// init traj filter
m_jnt3OTG.init(m_cmdJntPos[3], 0, m_retractVel, m_retractAcc, g_slaveArmCtrlCycleTime);

// set wait time before start retract
IF SlaveArmControl.m_slaveRobot.m_lastSlaveArmState[i_slaveArm.armIdx] = SlaveArmState_PanelReady THEN
	m_waitTime := 0;
ELSE
	m_waitTime :=1.0;
END_IF

// decide instrument joint zero position and init traj filter
FOR i:=1 TO 5 DO
	cycleNum := FLOOR(i_slaveArm.curJntPos[i+3]/g_2pi);
	m_instruJntTargetPos[i]:=cycleNum* g_2Pi;
	m_instruJntOTG[i].init(m_cmdJntPos[i+3], 0,m_instruJntVel, m_instruJntAcc, g_slaveArmCtrlCycleTime);
END_FOR

// update commands to arm
copyCmds(r_slaveArmCtrlCmd);
END_METHOD

END_FUNCTION_BLOCK

// ---- FBs_SlaveControllers/FB_SlaveCtrlInstruInvasion.TcPOU
// Brief: Slave Arm Invase instrument to record position
FUNCTION_BLOCK PUBLIC FB_SlaveCtrlInstruInvasion EXTENDS FB_SlaveArmCtrlBase
VAR_INPUT
END_VAR
VAR_OUTPUT
END_VAR
VAR
	// invasion buffer
	m_instruInvasionDepthSafetyBuffer :LREAL:= 0.01;
		
	// max damping when reaching invasion depth
	m_maxDamp :LREAL :=500;
	
	// current distance form target invasion depth 
	m_invasionDis :LREAL :=0;
	
	// distance threshold from target depth to start enable damp
	m_dampDisThres :LREAL :=0.03;
	
END_VAR

// override this function in each exact controller
METHOD PROTECTED calcCmdJntPos : BOOL
VAR_IN_OUT CONSTANT
	i_endoscopePose : ST_Frame;
	i_masterStatus :ST_MasterStatus;
	i_setupStatus: ST_SetupStatus;
	i_slaveArm :FB_SlaveArm;
END_VAR

VAR 
	curInstruDepth:LREAL;
END_VAR
m_cmdJntPos[3]:=i_slaveArm.curJntPos[3];
// compute current instrument depth
curInstruDepth := i_slaveArm.curJntPos[3]-i_slaveArm.instrument.instruTypeInfo.m_rodLength-i_slaveArm.instrument.instruTypeInfo.m_headLength
						- i_slaveArm.instrument.instruTypeInfo.m_fingerLength-m_instruInvasionDepthSafetyBuffer;

m_invasionDis:=curInstruDepth-i_slaveArm.m_instruInvasionDepth;
						
m_isFinished := curInstruDepth<= i_slaveArm.m_instruInvasionDepth;
END_METHOD

// override this function in each exact controller
METHOD PROTECTED calcCmdJntTrq : BOOL
VAR_IN_OUT CONSTANT
	i_endoscopePose : ST_Frame;
	i_masterStatus :ST_MasterStatus;
	i_setupStatus: ST_SetupStatus;
	i_slaveArm :FB_SlaveArm;
END_VAR
VAR
	dampScale :lreal ;
END_VAR
// set joint torque to zero in default
m_cmdJntTrq := g_zeroVec8d;

dampScale  :=LIMIT(0, 1-m_invasionDis/m_dampDisThres,1);
m_cmdJntTrq[3]:= -dampScale * m_maxDamp * i_slaveArm.curJntVel[3];
END_METHOD

METHOD PUBLIC init : BOOL
VAR_IN_OUT CONSTANT
	i_slaveArm	:FB_SlaveArm;
END_VAR
VAR_IN_OUT 
	r_slaveArmCtrlCmd :ST_SlaveArmCtrlCmds;
END_VAR
// check if to hold the command joint position unchanged
m_holdLastCmds := checkToHoldLastCmds(i_slaveArm);

//init
SUPER^.Init(i_slaveArm,r_slaveArmCtrlCmd);
m_invasionDis:=m_dampDisThres;

// only joint 3 is allowed to be pushed
m_jntOPMode := g_slaveAllPosMode;
m_jntOPMode[3]:=DriverOPMode_Trq;

// update commands to arm
copyCmds(r_slaveArmCtrlCmd);
END_METHOD

END_FUNCTION_BLOCK

// ---- FBs_SlaveControllers/FB_SlaveCtrlDisable.TcPOU
// Brief: Disable a Slave Arm 
FUNCTION_BLOCK PUBLIC FB_SlaveCtrlDisable EXTENDS FB_SlaveArmCtrlBase
VAR_INPUT
END_VAR
VAR_OUTPUT
END_VAR
VAR
END_VAR

// override this function in each exact controller
METHOD PROTECTED calcCmdJntPos : BOOL
VAR_IN_OUT CONSTANT
	// endoscope pose in cart coordinate
	i_endoscopePose : ST_Frame;
	
	// master arm data
	i_masterStatus :ST_MasterStatus;
	
	// setup arm data
	i_setupStatus: ST_SetupStatus;
	
	// slave arm data
	i_slaveArm :FB_SlaveArm;
END_VAR
m_cmdJntPos := i_slaveArm.curJntPos;
END_METHOD

// override this function in each exact controller
// NOTICE: set joint control mode here, and do some initialization if needed
METHOD PUBLIC init : BOOL
VAR_IN_OUT CONSTANT
	i_slaveArm	:FB_SlaveArm;
END_VAR
VAR_IN_OUT 
	r_slaveArmCtrlCmd :ST_SlaveArmCtrlCmds;
END_VAR


VAR
	i:INT;
END_VAR
SUPER^.Init(i_slaveArm,r_slaveArmCtrlCmd);

// disable all joints
 m_jntEnableFlag :=g_zeroVec8i;
 
 // update commands to arm
copyCmds(r_slaveArmCtrlCmd);
END_METHOD

END_FUNCTION_BLOCK

// ---- FBs_SlaveControllers/FB_SlaveCtrlInstruCali.TcPOU
// Brief: Calibrate the zero position of Instrument
FUNCTION_BLOCK PUBLIC FB_SlaveCtrlInstruCali EXTENDS FB_SlaveArmCtrlBase
VAR
	// mount motion planning
	m_jntOTG :ARRAY[1..8] OF FB_secOrdTrajFilter;
	m_instruMountVel :LREAL := 1*PI;
	m_instruMountAcc :LREAL := 2*PI;
	
	// 	cali status
	m_rollJntCaliStatus :INT := 0;
	m_pitchJntCaliStatus :INT := 0;
	m_yawJntCaliStatus :INT := 0;
	
	// flag if zero position is written to CoE
	m_zeroPosWritten :BOOL;
	
	// joint current threshold which indicate panel is buckled with instrument
	m_maxJntCurrent :LREAL := 100;
	
	// joint current threshold which indicate finger closed
	m_fingerCloseCurrent :LREAL := 50;
	
	// joint position at limits
	m_jntLimitPos1, m_jntLimitPos2, m_jntCaliPos :LREAL;
	m_jntLimitPos3, m_jntLimitPos4 :LREAL;

	// flag if joint is mounted
	m_jointMounted :ARRAY[1..8] OF BOOL := [5(FALSE)];
	
	// instrument mount motion range
	m_mountMotionAng :LREAL :=30*g_deg2Rad;
	
	// command mount motion
	m_targetMountPos :Vec8d;
	
	// instrument zero position
	m_instruZeroPosition :Vec5d;
	
	// angle to close finger
	m_baseCloseAngle :LREAL := 1*g_deg2Rad;
	m_bipolarCloseAngle :LREAL := 5*g_deg2Rad;
	m_proGraspCloseAngle:LREAL := 25*g_deg2Rad;
	
END_VAR

// override this function in each exact controller
METHOD PROTECTED calcCmdJntPos : BOOL
VAR_IN_OUT CONSTANT
	i_endoscopePose : ST_Frame;
	i_masterStatus :ST_MasterStatus;
	i_setupStatus: ST_SetupStatus;
	i_slaveArm :FB_SlaveArm;
END_VAR

VAR 
	i :INT;
END_VAR
// retur directly if instrument/endoscope is not readed
IF NOT i_slaveArm.instrument.onChipData.m_InstruReadSucceed THEN
	m_rollJntCaliStatus :=0;
	m_pitchJntCaliStatus :=0;
	m_yawJntCaliStatus :=0;
	m_zeroPosWritten :=FALSE;
	FOR i:=4 TO 8 DO
		m_jointMounted[i]:=FALSE;
	END_FOR
	return;
END_IF

// write zero position to CoE
IF m_yawJntCaliStatus = -1 THEN
	IF   NOT m_zeroPosWritten THEN
		m_zeroPosWritten := i_slaveArm.instrument.writeZeroPosToChip(m_instruZeroPosition[1],m_instruZeroPosition[2],m_instruZeroPosition[3]);
	END_IF
	RETURN;
END_IF;

// move joint to zero position
IF m_rollJntCaliStatus <> -1 THEN
	rollJntCali(i_slaveArm);
ELSIF m_pitchJntCaliStatus <> -1 THEN
	pitchJntCali(i_slaveArm);
ELSIF m_yawJntCaliStatus <> -1 THEN
	IF  i_slaveArm.instrument.InstruTypeInfo.m_isSingleFinger THEN
		yawJntCali_finger(i_slaveArm);
	ELSE
		yawJntCali_gripper(i_slaveArm);
	END_IF

END_IF

IF m_yawJntCaliStatus = -1 THEN
	FOR  i:=1 TO  5 DO
		m_instruZeroPosition[i]:=i_slaveArm.linkSingle[i+3];
	END_FOR
END_IF
END_METHOD

METHOD PUBLIC init : BOOL
VAR_IN_OUT CONSTANT
	i_slaveArm	:FB_SlaveArm;
END_VAR
VAR_IN_OUT 
	r_slaveArmCtrlCmd :ST_SlaveArmCtrlCmds;
END_VAR

VAR
	i : INT;
END_VAR
// check if to hold the command joint position unchanged
m_holdLastCmds := checkToHoldLastCmds(i_slaveArm);

SUPER^.Init(i_slaveArm,r_slaveArmCtrlCmd);
m_jntOPMode[4] := DriverOPMode_PosTrq;
m_jntOPMode[5] := DriverOPMode_PosTrq;
m_jntOPMode[6] := DriverOPMode_PosTrq;
m_jntOPMode[7] := DriverOPMode_PosTrq;
m_jntOPMode[8] := DriverOPMode_PosTrq;

FOR i:=4 TO 8 DO
	m_targetMountPos[i]:=m_cmdJntPos[i];
	m_jntOTG[i].init(m_targetMountPos[i], 0,m_instruMountVel, m_instruMountAcc, g_slaveArmCtrlCycleTime);
	m_jointMounted[i]:=FALSE;
END_FOR

m_rollJntCaliStatus :=0;
m_pitchJntCaliStatus :=0;
m_yawJntCaliStatus :=0;
m_zeroPosWritten := false;

// update commands to arm
copyCmds(r_slaveArmCtrlCmd);
END_METHOD

METHOD pitchJntCali : BOOL
VAR_IN_OUT CONSTANT
	i_slaveArm :FB_SlaveArm;
END_VAR

VAR 
	i :INT;
	curJntPos :Vec8d;
	jntIdx :INT;
END_VAR
jntIdx:=6;
curJntPos := i_slaveArm.curJntPos;

CASE m_pitchJntCaliStatus OF
	// rotate clockwise
	0:
		m_targetMountPos[jntIdx]:=curJntPos[jntIdx]+m_mountMotionAng;
	
		//buckle joint
		IF i_slaveArm.filtJntCurrent[jntIdx]> m_maxJntCurrent THEN 
			m_jntLimitPos1 := curJntPos[jntIdx];
			m_targetMountPos[jntIdx]:=curJntPos[jntIdx];
			m_jntOTG[jntIdx].init(m_targetMountPos[jntIdx], 0,m_instruMountVel, m_instruMountAcc, g_slaveArmCtrlCycleTime);
			m_pitchJntCaliStatus := 1;
		END_IF
		
	// rotate anticlockwise
	1:
		m_targetMountPos[jntIdx]:=curJntPos[jntIdx]-m_mountMotionAng;
	
		//buckle  joint
		IF i_slaveArm.filtJntCurrent[jntIdx]<- m_maxJntCurrent THEN 
			m_jntLimitPos2 := curJntPos[jntIdx];
			m_targetMountPos[jntIdx]:=curJntPos[jntIdx];
			m_jntOTG[jntIdx].init(m_targetMountPos[jntIdx], 0,m_instruMountVel, m_instruMountAcc, g_slaveArmCtrlCycleTime);
			m_pitchJntCaliStatus := 2;
		END_IF
	
	2:// calculate center/calibarted position
		m_targetMountPos[jntIdx] :=  (m_jntLimitPos1 + m_jntLimitPos2)/2+ i_slaveArm.instrument.instruTypeInfo.m_instruPitchBachlash/2.0;
		m_pitchJntCaliStatus := 3;

	3:
		IF ABS(m_targetMountPos[jntIdx]-curJntPos[jntIdx]) <GVL_SlaveControlParameters.g_jntCtrlAngTolHigh  THEN
			m_pitchJntCaliStatus := -1;
		END_IF
		
END_CASE

// traj plan
m_jntOTG[jntIdx].run(m_targetMountPos[jntIdx],0.0, o_cmdAcc=>m_cmdJntAcc[jntIdx],o_cmdVel=>m_cmdJntVel[jntIdx],o_cmdPos=>m_cmdJntPos[jntIdx]);
END_METHOD

METHOD rollJntCali : BOOL
VAR_IN_OUT CONSTANT
	i_slaveArm :FB_SlaveArm;
END_VAR

VAR 
	i :INT;
	curJntPos :Vec8d;
	jntIdx :INT;
END_VAR
jntIdx:=7;
curJntPos := i_slaveArm.curJntPos;

CASE m_rollJntCaliStatus OF
	// rotate clockwise
	0:
		m_targetMountPos[jntIdx]:=curJntPos[jntIdx]+m_mountMotionAng;
	
		//buckle  joint
		IF i_slaveArm.filtJntCurrent[jntIdx]> m_maxJntCurrent AND ABS(i_slaveArm.curJntVel[jntIdx]) < 1*g_deg2rad  THEN 
			m_jntLimitPos1 := curJntPos[jntIdx];
			m_targetMountPos[jntIdx]:=curJntPos[jntIdx];
			m_jntOTG[jntIdx].init(m_targetMountPos[jntIdx], 0,m_instruMountVel, m_instruMountAcc, g_slaveArmCtrlCycleTime);
			m_rollJntCaliStatus := 1;
		END_IF
		
	// rotate anticlockwise
	1:
		m_targetMountPos[jntIdx]:=curJntPos[jntIdx]-m_mountMotionAng;
	
		//buckle  joint
		IF i_slaveArm.filtJntCurrent[jntIdx]<- m_maxJntCurrent AND ABS(i_slaveArm.curJntVel[jntIdx]) < 1*g_deg2rad   THEN 
			m_jntLimitPos2 := curJntPos[jntIdx];
			m_targetMountPos[jntIdx]:=curJntPos[jntIdx];
			m_jntOTG[jntIdx].init(m_targetMountPos[jntIdx], 0,m_instruMountVel, m_instruMountAcc, g_slaveArmCtrlCycleTime);
			m_rollJntCaliStatus := 2;
		END_IF
	
	2:// calculate center/calibarted positio
		m_targetMountPos[jntIdx] :=  (m_jntLimitPos1 + m_jntLimitPos2)/2;
		m_rollJntCaliStatus := 3;

	3:
		IF ABS(m_targetMountPos[jntIdx]-curJntPos[jntIdx]) <GVL_SlaveControlParameters.g_jntCtrlAngTolHigh  THEN
			m_rollJntCaliStatus := -1;
		END_IF
		
END_CASE

// traj plan
m_jntOTG[jntIdx].run(m_targetMountPos[jntIdx],0.0, o_cmdAcc=>m_cmdJntAcc[jntIdx],o_cmdVel=>m_cmdJntVel[jntIdx],o_cmdPos=>m_cmdJntPos[jntIdx]);
END_METHOD

METHOD yawJntCali_finger : BOOL
VAR_IN_OUT CONSTANT
	i_slaveArm :FB_SlaveArm;
END_VAR

VAR 
	i :INT;
	curJntPos :Vec8d;
	jntIdx :INT;
END_VAR
jntIdx:=5;
curJntPos := i_slaveArm.curJntPos;

CASE m_yawJntCaliStatus OF
	// rotate clockwise
	0:
		m_targetMountPos[jntIdx]:=curJntPos[jntIdx]+m_mountMotionAng;
	
		//buckle  joint
		IF i_slaveArm.filtJntCurrent[jntIdx]> m_maxJntCurrent THEN 
			m_jntLimitPos1 := curJntPos[jntIdx];
			m_targetMountPos[jntIdx]:=curJntPos[jntIdx];
			m_jntOTG[jntIdx].init(m_targetMountPos[jntIdx], 0,m_instruMountVel, m_instruMountAcc, g_slaveArmCtrlCycleTime);
			m_yawJntCaliStatus := 1;
		END_IF
		
	// rotate anticlockwise
	1:
		m_targetMountPos[jntIdx]:=curJntPos[jntIdx]-m_mountMotionAng;
	
		//buckle  joint
		IF i_slaveArm.filtJntCurrent[jntIdx]<- m_maxJntCurrent THEN 
			m_jntLimitPos2 := curJntPos[jntIdx];
			m_targetMountPos[jntIdx]:=curJntPos[jntIdx];
			m_jntOTG[jntIdx].init(m_targetMountPos[jntIdx], 0,m_instruMountVel, m_instruMountAcc, g_slaveArmCtrlCycleTime);
			m_yawJntCaliStatus := 2;
		END_IF
	
	2:// calculate center/calibarted positio
		m_targetMountPos[jntIdx] :=  (m_jntLimitPos1 + m_jntLimitPos2)/2+i_slaveArm.instrument.instruTypeInfo.m_instruYawBacklash/2.0;;
		m_yawJntCaliStatus := 3;

	3:
		IF ABS(m_targetMountPos[jntIdx]-curJntPos[jntIdx]) <GVL_SlaveControlParameters.g_jntCtrlAngTolLow  THEN
			m_yawJntCaliStatus := -1;
		END_IF
		
END_CASE

// traj plan
m_jntOTG[jntIdx].run(m_targetMountPos[jntIdx],0.0, o_cmdAcc=>m_cmdJntAcc[jntIdx],o_cmdVel=>m_cmdJntVel[jntIdx],o_cmdPos=>m_cmdJntPos[jntIdx]);
END_METHOD

METHOD yawJntCali_gripper : BOOL
VAR_IN_OUT CONSTANT
	i_slaveArm :FB_SlaveArm;
END_VAR

VAR 
	curJntPos :Vec8d;
	gripCloseAng:LREAL;
END_VAR
curJntPos := i_slaveArm.curJntPos;

// determin finger close angle
IF i_slaveArm.instrument.instruType = InstruType_MarylandForceps OR i_slaveArm.instrument.instruType = InstruType_FenestratedForceps
	OR i_slaveArm.instrument.instruType = InstruType_CurvedBipolarDissector OR i_slaveArm.instrument.instruType = InstruType_MicroBipolarForceps THEN
	gripCloseAng := m_bipolarCloseAngle;
ELSIF i_slaveArm.instrument.instruType = InstruType_ProGraspForceps OR i_slaveArm.instrument.instruType = InstruType_ForceBipolar THEN
	gripCloseAng := m_proGraspCloseAngle;
ELSE
	gripCloseAng := m_baseCloseAngle;
END_IF

CASE m_yawJntCaliStatus OF
	// buckle joint4 and joint5 by moving toward limit
	0:
		//buckle panel with instrument
		// check if buckled 
		IF i_slaveArm.filtJntCurrent[4]<- m_maxJntCurrent THEN 
			m_jointMounted[4]:=TRUE;
			m_targetMountPos[4]:=curJntPos[4];
			m_jntOTG[4].init(m_targetMountPos[4], 0,m_instruMountVel, m_instruMountAcc, g_slaveArmCtrlCycleTime);
		END_IF
		IF i_slaveArm.filtJntCurrent[5]<- m_maxJntCurrent THEN 
			m_jointMounted[5]:=TRUE;
			m_targetMountPos[5]:=curJntPos[5];
			m_jntOTG[5].init(m_targetMountPos[5], 0,m_instruMountVel, m_instruMountAcc, g_slaveArmCtrlCycleTime);
		END_IF
		
		// set target joint position
		IF FALSE = m_jointMounted[4] THEN
			m_targetMountPos[4]:=curJntPos[4]-m_mountMotionAng;
		END_IF
		IF FALSE = m_jointMounted[5] THEN
			m_targetMountPos[5]:=curJntPos[5]-m_mountMotionAng;
		END_IF

		IF m_jointMounted[4] AND m_jointMounted[5] THEN
			m_yawJntCaliStatus := 1;
			m_jointMounted[4]:=FALSE;
			m_jointMounted[5]:=FALSE;
		END_IF
	// close finger
	1:
		//buckle panel with instrument
		// check if buckled 
		IF i_slaveArm.filtJntCurrent[4]> m_maxJntCurrent THEN 
			m_jointMounted[4]:=TRUE;
			m_targetMountPos[4]:=curJntPos[4];
			m_jntOTG[4].init(m_targetMountPos[4], 0,m_instruMountVel, m_instruMountAcc, g_slaveArmCtrlCycleTime);
		END_IF
		IF i_slaveArm.filtJntCurrent[5]> m_maxJntCurrent THEN 
			m_jointMounted[5]:=TRUE;
			m_targetMountPos[5]:=curJntPos[5];
			m_jntOTG[5].init(m_targetMountPos[5], 0,m_instruMountVel, m_instruMountAcc, g_slaveArmCtrlCycleTime);
		END_IF
		
		// set target joint position
		IF FALSE = m_jointMounted[4] THEN
			m_targetMountPos[4]:=curJntPos[4]+m_mountMotionAng;
		END_IF
		IF FALSE = m_jointMounted[5] THEN
			m_targetMountPos[5]:=curJntPos[5]+m_mountMotionAng;
		END_IF

		IF m_jointMounted[4] AND m_jointMounted[5] THEN
			m_yawJntCaliStatus := 2;
			m_jointMounted[4]:=FALSE;
			m_jointMounted[5]:=FALSE;
		END_IF
		
	2:// move joint5 to open gripper
		m_targetMountPos[4] := curJntPos[4]-i_slaveArm.instrument.instruTypeInfo.m_maxGripAngle/4.0;
		m_targetMountPos[5] := curJntPos[5]-i_slaveArm.instrument.instruTypeInfo.m_maxGripAngle/4.0;
		m_yawJntCaliStatus := 3;

	3:
		IF ABS(m_targetMountPos[5]-curJntPos[5]) <GVL_SlaveControlParameters.g_jntCtrlAngTolLow  THEN
			m_yawJntCaliStatus := 4;
		END_IF
			
	// roll clockwise to reach limit
	4:
		IF NOT(m_jointMounted[4]) THEN  
			// set target joint position
			m_targetMountPos[4]:=curJntPos[4]-m_mountMotionAng;
			// check if reach limit 
			IF i_slaveArm.filtJntCurrent[4]< -m_maxJntCurrent THEN 
				m_jointMounted[4]:=TRUE;
				m_jntLimitPos1 := curJntPos[4];
				m_targetMountPos[4]:=curJntPos[4];
				m_jntOTG[4].init(m_targetMountPos[4], 0,m_instruMountVel, m_instruMountAcc, g_slaveArmCtrlCycleTime);
			END_IF
		END_IF
		IF NOT(m_jointMounted[5]) THEN 
			// set target joint position
			m_targetMountPos[5]:=curJntPos[5]+m_mountMotionAng;
			// check if reach limit 
			IF i_slaveArm.filtJntCurrent[5]> m_maxJntCurrent THEN 
				m_jointMounted[5]:=TRUE;
				m_jntLimitPos2 := curJntPos[5];
				m_targetMountPos[5]:=curJntPos[5];
				m_jntOTG[5].init(m_targetMountPos[5], 0,m_instruMountVel, m_instruMountAcc, g_slaveArmCtrlCycleTime);
			END_IF	
		END_IF
		
		// transit
		IF m_jointMounted[4] AND m_jointMounted[5] THEN
			m_yawJntCaliStatus := 5;
			m_jointMounted[4]:=FALSE;
			m_jointMounted[5]:= FALSE;
		END_IF
		
	5:// move joint5 to open gripper
		m_targetMountPos[5] := curJntPos[5]-i_slaveArm.instrument.instruTypeInfo.m_maxGripAngle/2.0;
		m_yawJntCaliStatus := 6;

	6:
		IF ABS(m_targetMountPos[5]-curJntPos[5]) <GVL_SlaveControlParameters.g_jntCtrlAngTolLow  THEN
			m_yawJntCaliStatus := 7;
		END_IF

	// roll anticlockwise to reach limit
	7:
		IF NOT(m_jointMounted[4]) THEN  
			// set target joint position
			m_targetMountPos[4]:=curJntPos[4]+m_mountMotionAng;
			// check if reach limit 
			IF i_slaveArm.filtJntCurrent[4]>m_maxJntCurrent THEN 
				m_jointMounted[4]:=TRUE;
				m_jntLimitPos3 := curJntPos[4];
				m_targetMountPos[4]:=curJntPos[4];
				m_jntOTG[4].init(m_targetMountPos[4], 0,m_instruMountVel, m_instruMountAcc, g_slaveArmCtrlCycleTime);
			END_IF
		END_IF
		IF NOT(m_jointMounted[5]) THEN 
			// set target joint position
			m_targetMountPos[5]:=curJntPos[5]-m_mountMotionAng;
			// check if reach limit 
			IF i_slaveArm.filtJntCurrent[5]<- m_maxJntCurrent THEN 
				m_jointMounted[5]:=TRUE;
				m_jntLimitPos4 := curJntPos[5];
				m_targetMountPos[5]:=curJntPos[5];
				m_jntOTG[5].init(m_targetMountPos[5], 0,m_instruMountVel, m_instruMountAcc, g_slaveArmCtrlCycleTime);
			END_IF	
		END_IF
		
		// transit
		IF m_jointMounted[4] AND m_jointMounted[5] THEN
			m_yawJntCaliStatus := 8;
			m_jointMounted[4]:=FALSE;
			m_jointMounted[5]:= FALSE;
		END_IF
		
	8:// calculate center/calibarted position
		m_targetMountPos[4] := (m_jntLimitPos1 + m_jntLimitPos3)/2-i_slaveArm.instrument.instruTypeInfo.m_instruYawBacklash/2.0;
		m_targetMountPos[5] := (m_jntLimitPos2 + m_jntLimitPos4)/2+i_slaveArm.instrument.instruTypeInfo.m_instruYawBacklash/2.0;
		m_yawJntCaliStatus := 9;

	9:
		IF ABS(m_targetMountPos[4]-curJntPos[4]) <GVL_SlaveControlParameters.g_jntCtrlAngTolLow  AND
			ABS(m_targetMountPos[5]-curJntPos[5]) <GVL_SlaveControlParameters.g_jntCtrlAngTolLow  THEN
			m_targetMountPos[4] := curJntPos[4]+i_slaveArm.instrument.instruTypeInfo.m_instruYawBacklash;
			m_yawJntCaliStatus := 10;
		END_IF
		
	// close finger	
	10:
		IF ABS(m_targetMountPos[4]-curJntPos[4]) <GVL_SlaveControlParameters.g_jntCtrlAngTolLow  AND
			ABS(m_targetMountPos[5]-curJntPos[5]) <GVL_SlaveControlParameters.g_jntCtrlAngTolLow  THEN
				m_targetMountPos[4] := curJntPos[4]+gripCloseAng;
				m_targetMountPos[5] := curJntPos[5]+gripCloseAng;
			m_yawJntCaliStatus := 11;
		END_IF
		

	11:
		IF ABS(m_targetMountPos[4]-curJntPos[4]) <GVL_SlaveControlParameters.g_jntCtrlAngTolLow  AND
			ABS(m_targetMountPos[5]-curJntPos[5]) <GVL_SlaveControlParameters.g_jntCtrlAngTolLow  THEN
			m_yawJntCaliStatus := -1;
		END_IF

END_CASE

// traj plan
m_jntOTG[4].run(m_targetMountPos[4],0.0, o_cmdAcc=>m_cmdJntAcc[4],o_cmdVel=>m_cmdJntVel[4],o_cmdPos=>m_cmdJntPos[4]);
m_jntOTG[5].run(m_targetMountPos[5],0.0, o_cmdAcc=>m_cmdJntAcc[5],o_cmdVel=>m_cmdJntVel[5],o_cmdPos=>m_cmdJntPos[5]);
END_METHOD

END_FUNCTION_BLOCK

// ---- FBs_SlaveControllers/FB_SlaveCtrlScopeToggle.TcPOU
// Brief: toggle endoscope posture
FUNCTION_BLOCK PUBLIC FB_SlaveCtrlScopeToggle EXTENDS FB_SlaveArmCtrlBase
VAR_INPUT
END_VAR
VAR_OUTPUT
END_VAR
VAR
	// target joint position
	m_targetRotJntPos :LREAL;
	
	// motion planning
	m_jntOTG : FB_secOrdTrajFilter;
	m_rotVel :LREAL := 2*pi;
	m_rotAcc :LREAL := 6*pi;
	
END_VAR

// override this function in each exact controller
METHOD PROTECTED calcCmdJntPos : BOOL
VAR_IN_OUT CONSTANT
	i_endoscopePose : ST_Frame;
	i_masterStatus :ST_MasterStatus;
	i_setupStatus: ST_SetupStatus;
	i_slaveArm :FB_SlaveArm;
END_VAR

VAR 
	i :INT;
	trackErr:LREAL;
END_VAR
// traj plan
m_jntOTG.run(m_targetRotJntPos, 0.0, o_cmdAcc=>m_cmdJntAcc[8],o_cmdVel=>m_cmdJntVel[8],o_cmdPos=>m_cmdJntPos[8]);

// joint6 output torque to help rotation motion
IF m_jntOPMode[6] = DriverOPMode_Trq THEN
	m_cmdJntTrq[6] := -0.5*i_slaveArm.cmdJntTrq[7];
END_IF

// reach target check
trackErr := ABS(i_slaveArm.curJntPos[8] - m_targetRotJntPos);
m_isFinished := trackErr <2*g_jntCtrlAngTolHigh AND i_slaveArm.curJntVel[8]<g_jntStaticVelThres;
END_METHOD

METHOD PUBLIC init : BOOL
VAR_IN_OUT CONSTANT
	i_slaveArm	:FB_SlaveArm;
END_VAR
VAR_IN_OUT 
	r_slaveArmCtrlCmd :ST_SlaveArmCtrlCmds;
END_VAR

VAR
	i:INT;
	cycleNum:LREAL;
END_VAR
// check if to hold the command joint position unchanged
m_holdLastCmds := checkToHoldLastCmds(i_slaveArm);

SUPER^.Init(i_slaveArm,r_slaveArmCtrlCmd);
m_jntOPMode[6] := DriverOPMode_PosTrq;
m_jntOPMode[7] := DriverOPMode_PosTrq;
m_jntOPMode[8] := DriverOPMode_PosTrq;

// endoscope posture toggle
IF i_slaveArm.instrument.nextScopePosture <> i_slaveArm.instrument.curScopePosture AND i_slaveArm.instrument.curScopeType = EndoScopeType_30 THEN
	IF i_slaveArm.instrument.nextScopePosture = EndoScopePosture_HeadDown THEN
		m_targetRotJntPos := m_cmdJntPos[8] + PI/i_slaveArm.instrument.m_endoscopeRotateReduction;
	ELSE
		m_targetRotJntPos := m_cmdJntPos[8] - PI/i_slaveArm.instrument.m_endoscopeRotateReduction;
	END_IF
ELSE
	m_targetRotJntPos := m_cmdJntPos[8];
END_IF

// init traj filter
m_jntOTG.init(m_cmdJntPos[8], 0, m_rotVel, m_rotAcc, g_slaveArmCtrlCycleTime);

// update endoscope type/posture
i_slaveArm.instrument.curScopeType := i_slaveArm.instrument.nextScopeType;
i_slaveArm.instrument.curScopePosture := i_slaveArm.instrument.nextScopePosture;

// update commands to arm
copyCmds(r_slaveArmCtrlCmd);
END_METHOD

END_FUNCTION_BLOCK

// ---- FBs_SlaveControllers/FB_SlaveCtrlPerformance.TcPOU
// Brief: Slave Arm performance test
FUNCTION_BLOCK FB_SlaveCtrlPerformance EXTENDS FB_SlaveArmCtrlBase
VAR_INPUT
END_VAR
VAR_OUTPUT
END_VAR
VAR CONSTANT
	//Number of data recording points
	m_dataSum:INT:=8000;
END_VAR

VAR
	//test step
	m_testStep:INT:=-1;
	
	//test joint
	m_testJnt:INT;
	
	//trajectory planner
	m_caliTrajIdx: INT := 1;
	m_caliPlanner: ARRAY[1..4] OF FB_TrajMoveJ;
	m_caliPlannerStart: FB_TrajMoveJ;
	
	//speed test variable
	m_speedMaxTest:BOOL;
	
	//trajectory segment
	m_caliMotionSegs :INT :=4;
	m_graCaliTraj:ARRAY [1..4, 1..g_sJntNum] OF LREAL;
	
	//trajectory velocity/acceleration/jerk
	m_caliMaxjntVel:Vec8d:=[2(2.5*g_deg2Rad), 0.01, 5(2.5*g_deg2Rad)];
	m_caliMaxjntAcc:Vec8d:=[8(0.5)];
	m_caliMaxjntJerk:Vec8d:=[8(2.0)];
	
	//Extreme joint position
	m_minJntPos: ARRAY[1..g_sJntNum] OF LREAL;
	m_maxJntPos: ARRAY[1..g_sJntNum] OF LREAL;
	
	//data record idx
	i,j:INT;
	id,idx:INT;
	
	//Number of data recording points
	m_dataRecordNum_2,m_dataRecordNum_3:INT;
	
	//The current values of the second and third trajectories
	m_jntCurrentId2:ARRAY[1..m_dataSum,1..3] OF LREAL;
	m_jntCurrentId3:ARRAY[1..m_dataSum,1..3] OF LREAL;
	
	//sampling interval
	m_samplingInterval:INT:=80;
	
	//friction record value
	m_CoulombFriction,m_ViscousFriction:ARRAY[1..m_dataSum,1..3] OF LREAL;
	
	//friction summation
	m_CoulombFrictionSum,m_ViscousFrictionSum:ARRAY[1..3] OF LREAL;
	
	//friction averange
	m_CoulombFrictionAve,m_ViscousFrictionAve:ARRAY[1..3] OF LREAL;
	
	//friction maxmum value
	m_CoulombFrictionMax,m_ViscousFrictionMax:ARRAY[1..3] OF LREAL;
	
	//motion Frequency and angular frequency
	//m_Frequency:LREAL:=3; 	m_w:LREAL;
	m_Frequency:LREAL:=1; 	m_w:LREAL;
	
	//motion Frequency and angular frequency for speed test
	//m_FrequencySpeed:LREAL:=0.5; 	m_wSpeed:LREAL;
	m_FrequencySpeed:LREAL:=1; 	m_wSpeed:LREAL;
	
	//Dynamic performance testing time
	m_t:LREAL;
	
	//Dynamic performance testing motion range
	m_motionRange:ARRAY[1..3] OF LREAL:=[0.05,0.05,0.020];
	
	//Starting point for dynamic performance testing
	m_posOffset:ARRAY[1..g_sJntNum] OF LREAL;
	
	//Number of dynamic performance tests
	m_testNum:INT:=5;
	
	//motion range for maximum speed test
	m_motionRangeSpeed:ARRAY[1..3] OF LREAL:=[0.4,0.4,0.15];
	
	//initJntPos,startJntPos,endJntPos :Vec8d;
	initJntPos,startJntPos,endJntPos :Vec8d;
	
	//Motion amplitude and frequency
	m_motionAmplitude:ARRAY[1..3] OF LREAL;
	m_motionRadiusFre:LREAL;	
	m_Fre:LREAL;
	m_testTime:LREAL;
END_VAR

// override this function in each exact controller
METHOD PROTECTED calcCmdJntPos : BOOL
VAR_IN_OUT CONSTANT
	// endoscope pose in cart coordinate
	i_endoscopePose : ST_Frame;
	
	// master arm data
	i_masterStatus :ST_MasterStatus;
	
	// setup arm data
	i_setupStatus: ST_SetupStatus;
	
	// slave arm data
	i_slaveArm :FB_SlaveArm;
END_VAR


CASE m_testStep OF
	0: //test the motion range/joint friction/joint gap		
		IF m_caliPlanner[m_caliTrajIdx].isGene = FALSE THEN
			calcCmdJntPos:=FALSE;
			RETURN;
		END_IF
		
		// traj plan
		calcCmdJntPos :=m_caliPlanner[m_caliTrajIdx].evaluate(m_timePeriod, jntPos=> m_cmdJntPos, jntVel=>m_cmdJntVel, jntAcc=> m_cmdJntAcc);
		
		// check if to transit to next segment		
		IF(m_timePeriod > m_caliPlanner[m_caliTrajIdx].duration) THEN
			m_caliTrajIdx:=m_caliTrajIdx+1;
			m_timePeriod:=0;
			idx:=0;
			id:=0;
		END_IF
		
		// check if to terminated
		IF(m_caliTrajIdx > m_caliMotionSegs) THEN
			m_testStep:=10;
		END_IF
		
		//data record
		IF (m_caliTrajIdx=2) THEN
			//motion from joint min to joint max
			idx:=idx+1;
			IF (idx>=m_samplingInterval) THEN
				idx:=0;
				id:=id+1;
				m_dataRecordNum_2:=id;
				FOR j:=1 TO 3 BY 1 DO
					m_jntCurrentId2[id,j]:=i_slaveArm.filtJntCurrent[j]*gvl_SlaveMotorParameters.g_motorDir[j];
				END_FOR
			END_IF
		ELSIF (m_caliTrajIdx=3) THEN
			//motion from joint max to joint min
			idx:=idx+1;
			IF (idx>=m_samplingInterval) THEN
				idx:=0;
				id:=id+1;
				m_dataRecordNum_3:=id;
				FOR j:=1 TO 3 BY 1 DO
					m_jntCurrentId3[id,j]:=i_slaveArm.filtJntCurrent[j]*gvl_SlaveMotorParameters.g_motorDir[j];
				END_FOR
			END_IF
		END_IF
		
	
	10: //Process the data from the above steps				
		id:=0;		
		FOR i:=1 TO m_dataRecordNum_2 BY 1 DO
			idx:=(m_dataRecordNum_3-i)+1;
			IF (idx>0) THEN
				id:=id+1;  //Number of groups for recording data
				FOR j:=1 TO 3 BY 1 DO
					m_CoulombFriction[i,j]:=(m_jntCurrentId2[i,j]-m_jntCurrentId3[idx,j])/2;
					m_ViscousFriction[i,j]:=(m_jntCurrentId2[i,j]+m_jntCurrentId3[idx,j])/2;
					
					m_CoulombFrictionSum[j]:=m_CoulombFrictionSum[j]+m_CoulombFriction[i,j];
					m_ViscousFrictionSum[j]:=m_ViscousFrictionSum[j]+m_ViscousFriction[i,j];
					
					IF (m_CoulombFriction[i,j]>m_CoulombFrictionMax[j]) THEN
						m_CoulombFrictionMax[j]:=m_CoulombFriction[i,j];
					END_IF
					
					IF (m_ViscousFriction[i,j]>m_ViscousFrictionMax[j]) THEN
						m_ViscousFrictionMax[j]:=m_ViscousFriction[i,j];
					END_IF					
				END_FOR				
			END_IF			
		END_FOR
		
		FOR j:=1 TO 3 BY 1 DO
			m_CoulombFrictionAve[j]:=m_CoulombFrictionSum[j]/id;
			m_ViscousFrictionAve[j]:=m_ViscousFrictionSum[j]/id;
		END_FOR
		i:=1; m_t:=0;
		m_speedMaxTest:=FALSE;
		m_testStep:=20;
		
		
	20: //m_caliPlannerStart initialization		
		IF (m_speedMaxTest=FALSE) THEN
			m_motionAmplitude:=m_motionRange;
        	m_motionRadiusFre:=m_w;
			m_Fre:=m_Frequency;
		ELSE
			m_motionAmplitude:=m_motionRangeSpeed; 
			m_motionRadiusFre:=m_wSpeed;
			m_Fre:=m_FrequencySpeed;
		END_IF
		
		startJntPos:=i_slaveArm.curJntPos; 
		endJntPos:=m_posOffset;
		m_caliPlannerStart.init(startJntPos,endJntPos,m_caliMaxjntVel, m_caliMaxJntAcc, m_caliMaxJntJerk);
		m_timePeriod:=0;
		m_testStep:=30;
		
		
	30: //move to the start point
		IF m_caliPlannerStart.isGene = FALSE THEN
			calcCmdJntPos:=FALSE;
			RETURN;
		END_IF
		calcCmdJntPos :=m_caliPlannerStart.evaluate(m_timePeriod, jntPos=> m_cmdJntPos, jntVel=>m_cmdJntVel, jntAcc=> m_cmdJntAcc);			
		IF(m_timePeriod > m_caliPlannerStart.duration) THEN			
			m_timePeriod:=0;			
			m_testStep:=40;
		END_IF
			
		
	40: //Dynamic tracking capability test---3HZ
		m_t:=m_t+g_slaveArmCtrlCycleTime;
		sinusoidalMotion(posOffset:= endJntPos[i], amplitude:= m_motionAmplitude[i], t:= m_t, w:= m_motionRadiusFre, pos=> m_cmdJntPos[i], vel=> m_cmdJntVel[i], acc=> m_cmdJntAcc[i]);
		m_testTime:=(m_testNum+0.25)/m_Fre;
		
		IF (m_t>m_testTime) THEN
			m_cmdJntVel[i]:=0; 	m_cmdJntAcc[i]:=0;
			i:=i+1; 
			m_t:=0;
			m_testStep:=20;
			IF (i=4) AND (m_speedMaxTest=FALSE) THEN
				i:=1;
				m_speedMaxTest:=TRUE;
				m_testStep:=20;
			ELSIF (i=4) AND (m_speedMaxTest=TRUE) THEN
				i:=1;
				m_testStep:=-1;
				m_isFinished:=TRUE;
			END_IF
		END_IF			
	
		
	50: //
		

	-1: //
END_CASE
END_METHOD

// override this function in each exact controller
// NOTICE: set joint control mode here, and do some initialization if needed
METHOD PUBLIC init : BOOL
VAR_IN_OUT CONSTANT
	i_slaveArm	:FB_SlaveArm;
END_VAR
VAR_IN_OUT 
	r_slaveArmCtrlCmd :ST_SlaveArmCtrlCmds;
END_VAR
VAR
		//
END_VAR
SUPER^.Init(i_slaveArm,r_slaveArmCtrlCmd);
m_caliTrajIdx :=1;
m_jntOPMode := g_slaveAllPosTrqMode;


//joint position limit
m_minJntPos:=GVL_SlaveMotorParameters.g_minJntPos;
m_maxJntPos:=GVL_SlaveMotorParameters.g_maxJntPos;


//trajectory target position
FOR i:=1 TO 4 BY 1 DO
	FOR j:=1 TO 3 DO
		IF (i=1) THEN
			m_graCaliTraj[i,j]:=m_minJntPos[j];
		ELSIF (i=2) THEN
			m_graCaliTraj[i,j]:=m_maxJntPos[j];
		ELSIF (i=3) THEN
			m_graCaliTraj[i,j]:=m_minJntPos[j];
		ELSIF (i=4) THEN
			m_graCaliTraj[i,j]:=(m_minJntPos[j]+m_maxJntPos[j])/2;
		END_IF
	END_FOR
END_FOR


//first segment---move from the current position to the minimum value
initJntPos:=i_slaveArm.curJntPos;
startJntPos:=initJntPos;
endJntPos:=startJntPos;
FOR j:=1 TO 3 DO
	endJntPos[j]:=m_graCaliTraj[1,j];
END_FOR
m_caliPlanner[1].init(startJntPos,endJntPos,m_caliMaxjntVel, m_caliMaxJntAcc, m_caliMaxJntJerk);


// other segments
FOR i:=2 TO m_caliMotionSegs DO 
	startJntPos := endJntPos;
	endJntPos:=startJntPos;
	FOR j:=1 TO 3 DO
		endJntPos[j]:=m_graCaliTraj[i,j];
	END_FOR
	m_caliPlanner[i].init(startJntPos,endJntPos,m_caliMaxjntVel, m_caliMaxJntAcc, m_caliMaxJntJerk);
END_FOR


//reset the step
m_testStep:=0;


//motion frequency
m_w:=2.0*pi*m_Frequency;
m_wSpeed:=2.0*pi*m_FrequencySpeed;
vecAdd(m_maxJntPos,m_minJntPos,m_posOffset); vecSelfMultiNum(m_posOffset,0.5);


//Initialization of calculation results
FOR j:=1 TO 3 BY 1 DO
	m_CoulombFrictionSum[j]:=0; m_CoulombFrictionMax[j]:=0; m_CoulombFrictionAve[j]:=0;
	m_ViscousFrictionSum[j]:=0; m_ViscousFrictionMax[j]:=0; m_ViscousFrictionAve[j]:=0;
END_FOR


// update commands to arm
copyCmds(r_slaveArmCtrlCmd);
END_METHOD

METHOD sinusoidalMotion : BOOL
VAR_INPUT
	posOffset:LREAL;
	amplitude:LREAL;
	t:LREAL; //time
	w:LREAL; //angular frequency
END_VAR

VAR_OUTPUT
	pos:LREAL;
	vel:LREAL;
	acc:LREAL;
END_VAR

VAR
	
END_VAR

pos:=posOffset+amplitude*SIN(w*t);
vel:=amplitude*w*COS(w*t);
acc:=-amplitude*w*w*SIN(w*t);
END_METHOD

END_FUNCTION_BLOCK

// ---- FBs_SlaveControllers/FB_SlaveCtrlStop.TcPOU
// Brief: Slave Arm Joint1-3 decelerate to stop
FUNCTION_BLOCK PUBLIC FB_SlaveCtrlStop EXTENDS FB_SlaveArmCtrlBase
VAR
	// stop motion is terminated after set time period
	m_maxStopPeriod :LREAL := 0.12;
	
	// deceleration period 
	m_decPeriod :LREAL := 0.1;

END_VAR

// override this function in each exact controller
METHOD PROTECTED calcCmdJntPos : BOOL
VAR_IN_OUT CONSTANT
	i_endoscopePose : ST_Frame;
	i_masterStatus :ST_MasterStatus;
	i_setupStatus: ST_SetupStatus;
	i_slaveArm :FB_SlaveArm;
END_VAR

VAR 
	i :INT;
	nextCmdVel :LREAL;
END_VAR
IF m_isFinished THEN
	m_cmdJntVel := g_zeroVec8d;
	m_cmdJntPos := i_slaveArm.curJntPos;
	m_FFJntTrq := g_zeroVec8d;
	RETURN;
END_IF

IF m_timePeriod > m_maxStopPeriod  THEN
	m_isFinished := TRUE;
	RETURN;
END_IF

FOR i := 1 TO 3 DO
	IF m_timePeriod > m_decPeriod THEN
		m_cmdJntVel[i] := 0;
		m_FFJntTrq[i]:=0;
	ELSE
		nextCmdVel := m_cmdJntVel[i] + m_cmdJntAcc[i]*g_slaveArmCtrlCycleTime;
		m_cmdJntPos[i] := m_cmdJntPos[i] + (nextCmdVel + m_cmdJntVel[i])*g_slaveArmCtrlCycleTime/2.0;
		m_cmdJntVel[i] := nextCmdVel;
		m_FFJntTrq[i] :=  i_slaveArm.massMat[i,i] * m_cmdJntAcc[i] ;
	END_IF
END_FOR
END_METHOD

METHOD PUBLIC init : BOOL
VAR_IN_OUT CONSTANT
	i_slaveArm	:FB_SlaveArm;
END_VAR
VAR_IN_OUT 
	r_slaveArmCtrlCmd :ST_SlaveArmCtrlCmds;
END_VAR
VAR
	i:INT;
	maxJntTrq:LREAL;
END_VAR
SUPER^.Init(i_slaveArm,r_slaveArmCtrlCmd);

// determine joint deceleration
FOR i:=1 TO 3 DO 
	m_jntOPMode[i] := DriverOPMode_PosTrq;
	m_cmdJntVel[i] := i_slaveArm.curJntVel[i];
	i_slaveArm.m_jntPIDCtrl[i].reset();
	m_cmdJntAcc[i] := -i_slaveArm.curJntVel[i]/m_decPeriod;
END_FOR

// update commands to arm
copyCmds(r_slaveArmCtrlCmd);
END_METHOD

END_FUNCTION_BLOCK

// ---- SafetyCheck/ASSERT.TcPOU
// this function is used to check if input statament is true.
// if false, the code will trigger a zero-devide exception and stop the whole program by PLC
FUNCTION ASSERT : BOOL
VAR_INPUT
	statement:BOOL;
END_VAR
VAR
	zero:INT :=0;
	res :REAL:=0;
END_VAR

IF NOT(statement) THEN
	res := 1/zero;
END_IF

ASSERT := true;

END_FUNCTION

// ---- SafetyCheck/Fb_dataRecord.TcPOU
FUNCTION_BLOCK Fb_dataRecord 
VAR_INPUT
	
END_VAR
VAR_OUTPUT
END_VAR
VAR
	i,j,k,z,c:UDINT;
	Index:ARRAY[1..g_maxNum] OF INT:=[5(2)];
	m_Index:ARRAY[1..g_maxNum] OF UDINT;
	Err,Arm,Joint,ErrID:UDINT;
	ErrWritingFalg:ARRAY [1..g_maxNum] OF BOOL:=[5(FALSE)];
	ArrayErrCodeTypeLast:ARRAY [1..g_maxNum] OF UDINT;
	sPath: STRING(255);
	mErr:ARRAY [0..MAX_CSV_COLUMNS] OF STRING(255);
	StartRecord:ARRAY[1..g_maxNum] OF R_TRIG;
	RecordCompletion:ARRAY[1..g_maxNum] OF F_TRIG;
	errFlagDelay1s :ARRAY [1..g_maxNum] OF TON;
	ErrWritingAllowed :ARRAY [1..g_maxNum] OF BOOL:=[5(FALSE)];
	
	fbSysTime	: 	GETSYSTEMTIME;
	tFileTime	:	T_FILETIME;  
	
	_tNow,	_tNowBoLin	:	TIMESTRUCT; 
	fbFormat 	: 	FB_FormatString;
	_sPathFormat	: T_MaxString := '%s%d-%d-%d-%d-%d-%d-%s-%s-%s.csv'; 
	
	_iBuffer: UDINT := 1;
		
	StartTime:LREAL;
	
	iZeroRowsData:ARRAY[0..MAX_CSV_ROWS] OF  ARRAY [0..MAX_CSV_COLUMNS] OF STRING(MAX_CSV_FIELD_LENGTH);
	iZeroErrCode:ARRAY [1..g_maxNum] OF ARRAY[0..100] OF UDINT;
	gCSV_Buffer: ARRAY[1..MAX_CSV_RING_BUFFER] OF ST_Buffer;
	mErrNameLocation: ARRAY [1..MAX_CSV_RING_BUFFER,0..MAX_CSV_COLUMNS] OF STRING(MAX_CSV_FIELD_LENGTH);
END_VAR

METHOD armDataCast : BOOL
VAR_IN_OUT CONSTANT
	i_safetyCheckVar :ARRAY[1..g_maxNum] OF checkInputVariable;
	i_setupStatus : ST_SetupStatus;
	i_slaveStatus : ST_SlaveStatus;
	i_setupJointData : ST_SetupJointData;
	i_slaveJointData : ST_SlaveJointData;
END_VAR

FOR i:= 1 TO 4 BY 1 DO
	IF ErrWritingFalg[i] = FALSE THEN
	j:=1;
	//状态机
	gCSV_Buffer[i].aBuffer[Index[i]][j:=j+1]:=LREAL_TO_FMTSTR(i_setupStatus.m_armState[i],0, TRUE);  gCSV_Buffer[i].aBuffer[1][j]:='setupArmMachine';
	gCSV_Buffer[i].aBuffer[Index[i]][j:=j+1]:=LREAL_TO_FMTSTR(i_slaveStatus.m_armState[i],0, TRUE);  gCSV_Buffer[i].aBuffer[1][j]:='slaveArmMachine';
	
	//link pos
	gCSV_Buffer[i].aBuffer[Index[i]][j:=j+1]:=LREAL_TO_STRING(i_setupJointData.m_curLinkPos[i][3]);   gCSV_Buffer[i].aBuffer[1][j]:='curLinkPosJ3';
	gCSV_Buffer[i].aBuffer[Index[i]][j:=j+1]:=LREAL_TO_STRING(i_setupJointData.m_curLinkPos[i][4]);   gCSV_Buffer[i].aBuffer[1][j]:='curLinkPosJ4';
	gCSV_Buffer[i].aBuffer[Index[i]][j:=j+1]:=LREAL_TO_STRING(i_setupJointData.m_curLinkPos[i][5]);   gCSV_Buffer[i].aBuffer[1][j]:='curLinkPosJ5';
	gCSV_Buffer[i].aBuffer[Index[i]][j:=j+1]:=LREAL_TO_STRING(i_slaveJointData.m_curLinkPos[i][1]);   gCSV_Buffer[i].aBuffer[1][j]:='curLinkPosJ6';
	gCSV_Buffer[i].aBuffer[Index[i]][j:=j+1]:=LREAL_TO_STRING(i_slaveJointData.m_curLinkPos[i][2]); gCSV_Buffer[i].aBuffer[1][j]:='curLinkPosJ7';
	gCSV_Buffer[i].aBuffer[Index[i]][j:=j+1]:=LREAL_TO_STRING(i_slaveJointData.m_curLinkPos[i][3]); gCSV_Buffer[i].aBuffer[1][j]:='curLinkPosJ8';
	
	//motor pos / curJntPos
	gCSV_Buffer[i].aBuffer[Index[i]][j:=j+1]:=LREAL_TO_STRING(i_setupJointData.m_curJntPos[i][3]);  gCSV_Buffer[i].aBuffer[1][j]:='curJntPosJ3';
	gCSV_Buffer[i].aBuffer[Index[i]][j:=j+1]:=LREAL_TO_STRING(i_setupJointData.m_curJntPos[i][4]);  gCSV_Buffer[i].aBuffer[1][j]:='curJntPosJ4';
	gCSV_Buffer[i].aBuffer[Index[i]][j:=j+1]:=LREAL_TO_STRING(i_setupJointData.m_curJntPos[i][5]);  gCSV_Buffer[i].aBuffer[1][j]:='curJntPosJ5';
	gCSV_Buffer[i].aBuffer[Index[i]][j:=j+1]:=LREAL_TO_STRING(i_slaveJointData.m_curJntPos[i][1]);  gCSV_Buffer[i].aBuffer[1][j]:='curJntPosJ6';
	gCSV_Buffer[i].aBuffer[Index[i]][j:=j+1]:=LREAL_TO_STRING(i_slaveJointData.m_curJntPos[i][2]); gCSV_Buffer[i].aBuffer[1][j]:='curJntPosJ7';
	gCSV_Buffer[i].aBuffer[Index[i]][j:=j+1]:=LREAL_TO_STRING(i_slaveJointData.m_curJntPos[i][3]); gCSV_Buffer[i].aBuffer[1][j]:='curJntPosJ8';
	
	
	//target joint position 
	gCSV_Buffer[i].aBuffer[Index[i]][j:=j+1]:=LREAL_TO_STRING(i_setupJointData.m_cmdJntPos[i][3]);  gCSV_Buffer[i].aBuffer[1][j]:='cmdJntPosJ3';
	gCSV_Buffer[i].aBuffer[Index[i]][j:=j+1]:=LREAL_TO_STRING(i_setupJointData.m_cmdJntPos[i][4]);  gCSV_Buffer[i].aBuffer[1][j]:='cmdJntPosJ4';
	gCSV_Buffer[i].aBuffer[Index[i]][j:=j+1]:=LREAL_TO_STRING(i_setupJointData.m_cmdJntPos[i][5]);  gCSV_Buffer[i].aBuffer[1][j]:='cmdJntPosJ5';
	gCSV_Buffer[i].aBuffer[Index[i]][j:=j+1]:=LREAL_TO_STRING(i_slaveJointData.m_cmdJntPos[i][1]);  gCSV_Buffer[i].aBuffer[1][j]:='cmdJntPosJ6';
	gCSV_Buffer[i].aBuffer[Index[i]][j:=j+1]:=LREAL_TO_STRING(i_slaveJointData.m_cmdJntPos[i][2]);  gCSV_Buffer[i].aBuffer[1][j]:='cmdJntPosJ7';
	gCSV_Buffer[i].aBuffer[Index[i]][j:=j+1]:=LREAL_TO_STRING(i_slaveJointData.m_cmdJntPos[i][3]);  gCSV_Buffer[i].aBuffer[1][j]:='cmdJntPosJ8';
	
	
	//current joint velocity
	gCSV_Buffer[i].aBuffer[Index[i]][j:=j+1]:=LREAL_TO_STRING(i_setupJointData.m_curJntVel[i][3]);  gCSV_Buffer[i].aBuffer[1][j]:='curJntVelJ3';
	gCSV_Buffer[i].aBuffer[Index[i]][j:=j+1]:=LREAL_TO_STRING(i_setupJointData.m_curJntVel[i][4]);  gCSV_Buffer[i].aBuffer[1][j]:='curJntVelJ4';
	gCSV_Buffer[i].aBuffer[Index[i]][j:=j+1]:=LREAL_TO_STRING(i_setupJointData.m_curJntVel[i][5]);  gCSV_Buffer[i].aBuffer[1][j]:='curJntVelJ5';
	gCSV_Buffer[i].aBuffer[Index[i]][j:=j+1]:=LREAL_TO_STRING(i_slaveJointData.m_curJntVel[i][1]);  gCSV_Buffer[i].aBuffer[1][j]:='curJntVelJ6';
	gCSV_Buffer[i].aBuffer[Index[i]][j:=j+1]:=LREAL_TO_STRING(i_slaveJointData.m_curJntVel[i][2]);  gCSV_Buffer[i].aBuffer[1][j]:='curJntVelJ7';
	gCSV_Buffer[i].aBuffer[Index[i]][j:=j+1]:=LREAL_TO_STRING(i_slaveJointData.m_curJntVel[i][3]);  gCSV_Buffer[i].aBuffer[1][j]:='curJntVelJ8';
	
	//command arm pose
	gCSV_Buffer[i].aBuffer[Index[i]][j:=j+1]:=LREAL_TO_STRING(i_slaveStatus.m_cmdArmPose[i].m_pos[1]);  gCSV_Buffer[i].aBuffer[1][j]:='cmdArmPose1';
	gCSV_Buffer[i].aBuffer[Index[i]][j:=j+1]:=LREAL_TO_STRING(i_slaveStatus.m_cmdArmPose[i].m_pos[2]);  gCSV_Buffer[i].aBuffer[1][j]:='cmdArmPose2';
	gCSV_Buffer[i].aBuffer[Index[i]][j:=j+1]:=LREAL_TO_STRING(i_slaveStatus.m_cmdArmPose[i].m_pos[3]);  gCSV_Buffer[i].aBuffer[1][j]:='cmdArmPose3';
	//gCSV_Buffer[i].aBuffer[Index[i]][j:=j+1]:=LREAL_TO_STRING(i_slaveStatus.m_cmdArmPose[i].m_rot[1]);  gCSV_Buffer[i].aBuffer[1][j]:='cmdArmPose4';
	//gCSV_Buffer[i].aBuffer[Index[i]][j:=j+1]:=LREAL_TO_STRING(i_slaveStatus.m_cmdArmPose[i].m_rot[2]);  gCSV_Buffer[i].aBuffer[1][j]:='cmdArmPose5';
	//gCSV_Buffer[i].aBuffer[Index[i]][j:=j+1]:=LREAL_TO_STRING(i_slaveStatus.m_cmdArmPose[i].m_rot[3]);  gCSV_Buffer[i].aBuffer[1][j]:='cmdArmPose6';

	//current arm pose
	gCSV_Buffer[i].aBuffer[Index[i]][j:=j+1]:=LREAL_TO_STRING(i_slaveStatus.m_curArmPose[i].m_pos[1]);  gCSV_Buffer[i].aBuffer[1][j]:='curArmPose1';
	gCSV_Buffer[i].aBuffer[Index[i]][j:=j+1]:=LREAL_TO_STRING(i_slaveStatus.m_curArmPose[i].m_pos[2]);  gCSV_Buffer[i].aBuffer[1][j]:='curArmPose2';
	gCSV_Buffer[i].aBuffer[Index[i]][j:=j+1]:=LREAL_TO_STRING(i_slaveStatus.m_curArmPose[i].m_pos[3]);  gCSV_Buffer[i].aBuffer[1][j]:='curArmPose3';
	//gCSV_Buffer[i].aBuffer[Index[i]][j:=j+1]:=LREAL_TO_STRING(i_slaveStatus.m_curArmPose[i].m_rot[1]);  gCSV_Buffer[i].aBuffer[1][j]:='curArmPose4';
	//gCSV_Buffer[i].aBuffer[Index[i]][j:=j+1]:=LREAL_TO_STRING(i_slaveStatus.m_curArmPose[i].m_rot[2]);  gCSV_Buffer[i].aBuffer[1][j]:='curArmPose5';
	//gCSV_Buffer[i].aBuffer[Index[i]][j:=j+1]:=LREAL_TO_STRING(i_slaveStatus.m_curArmPose[i].m_rot[3]);  gCSV_Buffer[i].aBuffer[1][j]:='curArmPose6';
	
	//drive error word
	gCSV_Buffer[i].aBuffer[Index[i]][j:=j+1]:=UDINT_TO_STRING(i_safetyCheckVar[i].m_setupDriverInput[3].m_driverError);  gCSV_Buffer[i].aBuffer[1][j]:='driverErrorIOJ3'; 
	gCSV_Buffer[i].aBuffer[Index[i]][j:=j+1]:=UDINT_TO_STRING(i_safetyCheckVar[i].m_setupDriverInput[4].m_driverError);  gCSV_Buffer[i].aBuffer[1][j]:='driverErrorIOJ4'; 
	gCSV_Buffer[i].aBuffer[Index[i]][j:=j+1]:=UDINT_TO_STRING(i_safetyCheckVar[i].m_setupDriverInput[5].m_driverError);  gCSV_Buffer[i].aBuffer[1][j]:='driverErrorIOJ5'; 
	gCSV_Buffer[i].aBuffer[Index[i]][j:=j+1]:=UDINT_TO_STRING(i_safetyCheckVar[i].m_slaveDriverInput[1].m_driverError);  gCSV_Buffer[i].aBuffer[1][j]:='driverErrorIOJ6'; 
	gCSV_Buffer[i].aBuffer[Index[i]][j:=j+1]:=UDINT_TO_STRING(i_safetyCheckVar[i].m_slaveDriverInput[2].m_driverError); gCSV_Buffer[i].aBuffer[1][j]:='driverErrorIOJ7'; 
	gCSV_Buffer[i].aBuffer[Index[i]][j:=j+1]:=UDINT_TO_STRING(i_safetyCheckVar[i].m_slaveDriverInput[3].m_driverError); gCSV_Buffer[i].aBuffer[1][j]:='driverErrorIOJ8'; 
    
	//Electrical Angle deviation
	gCSV_Buffer[i].aBuffer[Index[i]][j:=j+1]:=DINT_TO_STRING(i_safetyCheckVar[i].m_setupDriverInput[3].m_electriAngleDev);  gCSV_Buffer[i].aBuffer[1][j]:='PhieErrIOJ3';
	gCSV_Buffer[i].aBuffer[Index[i]][j:=j+1]:=DINT_TO_STRING(i_safetyCheckVar[i].m_setupDriverInput[4].m_electriAngleDev);  gCSV_Buffer[i].aBuffer[1][j]:='PhieErrIOJ4';
	gCSV_Buffer[i].aBuffer[Index[i]][j:=j+1]:=DINT_TO_STRING(i_safetyCheckVar[i].m_setupDriverInput[5].m_electriAngleDev);  gCSV_Buffer[i].aBuffer[1][j]:='PhieErrIOJ5';
	gCSV_Buffer[i].aBuffer[Index[i]][j:=j+1]:=DINT_TO_STRING(i_safetyCheckVar[i].m_slaveDriverInput[1].m_electriAngleDev);  gCSV_Buffer[i].aBuffer[1][j]:='PhieErrIOJ6';
	gCSV_Buffer[i].aBuffer[Index[i]][j:=j+1]:=DINT_TO_STRING(i_safetyCheckVar[i].m_slaveDriverInput[2].m_electriAngleDev); gCSV_Buffer[i].aBuffer[1][j]:='PhieErrIOJ7';
	gCSV_Buffer[i].aBuffer[Index[i]][j:=j+1]:=DINT_TO_STRING(i_safetyCheckVar[i].m_slaveDriverInput[3].m_electriAngleDev); gCSV_Buffer[i].aBuffer[1][j]:='PhieErrIOJ8';
	
	
	//link encoder IO
	gCSV_Buffer[i].aBuffer[Index[i]][j:=j+1]:=DINT_TO_STRING(i_safetyCheckVar[i].m_setupDriverInput[3].m_linkEncoder);  gCSV_Buffer[i].aBuffer[1][j]:='curLinkIOJ3';
	gCSV_Buffer[i].aBuffer[Index[i]][j:=j+1]:=DINT_TO_STRING(i_safetyCheckVar[i].m_setupDriverInput[4].m_linkEncoder);  gCSV_Buffer[i].aBuffer[1][j]:='curLinkIOJ4';
	gCSV_Buffer[i].aBuffer[Index[i]][j:=j+1]:=DINT_TO_STRING(i_safetyCheckVar[i].m_setupDriverInput[5].m_linkEncoder);  gCSV_Buffer[i].aBuffer[1][j]:='curLinkIOJ5';
	gCSV_Buffer[i].aBuffer[Index[i]][j:=j+1]:=DINT_TO_STRING(i_safetyCheckVar[i].m_slaveDriverInput[1].m_linkEncoder);   gCSV_Buffer[i].aBuffer[1][j]:='curLinkIOJ6';
	gCSV_Buffer[i].aBuffer[Index[i]][j:=j+1]:=DINT_TO_STRING(i_safetyCheckVar[i].m_slaveDriverInput[2].m_linkEncoder); 	gCSV_Buffer[i].aBuffer[1][j]:='curLinkIOJ7';
	gCSV_Buffer[i].aBuffer[Index[i]][j:=j+1]:=DINT_TO_STRING(i_safetyCheckVar[i].m_slaveDriverInput[3].m_linkEncoder); 	gCSV_Buffer[i].aBuffer[1][j]:='curLinkIOJ8';
	
	//motor encoder  IO
	gCSV_Buffer[i].aBuffer[Index[i]][j:=j+1]:=DINT_TO_STRING(i_safetyCheckVar[i].m_setupDriverInput[3].m_motorEncoder);  gCSV_Buffer[i].aBuffer[1][j]:='curMotorEncIOJ3';
	gCSV_Buffer[i].aBuffer[Index[i]][j:=j+1]:=DINT_TO_STRING(i_safetyCheckVar[i].m_setupDriverInput[4].m_motorEncoder);  gCSV_Buffer[i].aBuffer[1][j]:='curMotorEncIOJ4';
	gCSV_Buffer[i].aBuffer[Index[i]][j:=j+1]:=DINT_TO_STRING(i_safetyCheckVar[i].m_setupDriverInput[5].m_motorEncoder);  gCSV_Buffer[i].aBuffer[1][j]:='curMotorEncIOJ5';
	gCSV_Buffer[i].aBuffer[Index[i]][j:=j+1]:=DINT_TO_STRING(i_safetyCheckVar[i].m_slaveDriverInput[1].m_motorEncoder);   gCSV_Buffer[i].aBuffer[1][j]:='curMotorEncIOJ6';
	gCSV_Buffer[i].aBuffer[Index[i]][j:=j+1]:=DINT_TO_STRING(i_safetyCheckVar[i].m_slaveDriverInput[2].m_motorEncoder); 	gCSV_Buffer[i].aBuffer[1][j]:='curMotorEncIOJ7';
	gCSV_Buffer[i].aBuffer[Index[i]][j:=j+1]:=DINT_TO_STRING(i_safetyCheckVar[i].m_slaveDriverInput[3].m_motorEncoder); 	gCSV_Buffer[i].aBuffer[1][j]:='curMotorEncIOJ8';
	
	//status word IO
	gCSV_Buffer[i].aBuffer[Index[i]][j:=j+1]:=UINT_TO_STRING(i_safetyCheckVar[i].m_setupDriverInput[3].m_statusWord);	gCSV_Buffer[i].aBuffer[1][j]:='statusWordIOJ3';
	gCSV_Buffer[i].aBuffer[Index[i]][j:=j+1]:=UINT_TO_STRING(i_safetyCheckVar[i].m_setupDriverInput[4].m_statusWord);	gCSV_Buffer[i].aBuffer[1][j]:='statusWordIOJ4';
	gCSV_Buffer[i].aBuffer[Index[i]][j:=j+1]:=UINT_TO_STRING(i_safetyCheckVar[i].m_setupDriverInput[5].m_statusWord);	gCSV_Buffer[i].aBuffer[1][j]:='statusWordIOJ5';
	gCSV_Buffer[i].aBuffer[Index[i]][j:=j+1]:=UINT_TO_STRING(i_safetyCheckVar[i].m_slaveDriverInput[1].m_statusWord);		gCSV_Buffer[i].aBuffer[1][j]:='statusWordIOJ6';
	gCSV_Buffer[i].aBuffer[Index[i]][j:=j+1]:=UINT_TO_STRING(i_safetyCheckVar[i].m_slaveDriverInput[2].m_statusWord);		gCSV_Buffer[i].aBuffer[1][j]:='statusWordIOJ7';
	gCSV_Buffer[i].aBuffer[Index[i]][j:=j+1]:=UINT_TO_STRING(i_safetyCheckVar[i].m_slaveDriverInput[3].m_statusWord);		gCSV_Buffer[i].aBuffer[1][j]:='statusWordIOJ8';

	//current torque IO
	gCSV_Buffer[i].aBuffer[Index[i]][j:=j+1]:=DINT_TO_STRING(i_safetyCheckVar[i].m_setupDriverInput[3].m_current);  gCSV_Buffer[i].aBuffer[1][j]:='curTorqueIOJ3';
	gCSV_Buffer[i].aBuffer[Index[i]][j:=j+1]:=DINT_TO_STRING(i_safetyCheckVar[i].m_setupDriverInput[4].m_current);  gCSV_Buffer[i].aBuffer[1][j]:='curTorqueIOJ4';
	gCSV_Buffer[i].aBuffer[Index[i]][j:=j+1]:=DINT_TO_STRING(i_safetyCheckVar[i].m_setupDriverInput[5].m_current);  gCSV_Buffer[i].aBuffer[1][j]:='curTorqueIOJ5';
	gCSV_Buffer[i].aBuffer[Index[i]][j:=j+1]:=DINT_TO_STRING(i_safetyCheckVar[i].m_slaveDriverInput[1].m_current);  gCSV_Buffer[i].aBuffer[1][j]:='curTorqueIOJ6';
	gCSV_Buffer[i].aBuffer[Index[i]][j:=j+1]:=DINT_TO_STRING(i_safetyCheckVar[i].m_slaveDriverInput[2].m_current);  gCSV_Buffer[i].aBuffer[1][j]:='curTorqueIOJ7';
	gCSV_Buffer[i].aBuffer[Index[i]][j:=j+1]:=DINT_TO_STRING(i_safetyCheckVar[i].m_slaveDriverInput[3].m_current);  gCSV_Buffer[i].aBuffer[1][j]:='curTorqueIOJ8';

	//target torque IO
	gCSV_Buffer[i].aBuffer[Index[i]][j:=j+1]:=DINT_TO_STRING(i_safetyCheckVar[i].m_setupDriverOutput[3].m_cmdCurrent);  gCSV_Buffer[i].aBuffer[1][j]:='cmdTorqueIOJ3';
	gCSV_Buffer[i].aBuffer[Index[i]][j:=j+1]:=DINT_TO_STRING(i_safetyCheckVar[i].m_setupDriverOutput[4].m_cmdCurrent);  gCSV_Buffer[i].aBuffer[1][j]:='cmdTorqueIOJ4';
	gCSV_Buffer[i].aBuffer[Index[i]][j:=j+1]:=DINT_TO_STRING(i_safetyCheckVar[i].m_setupDriverOutput[5].m_cmdCurrent);  gCSV_Buffer[i].aBuffer[1][j]:='cmdTorqueIOJ5';
	gCSV_Buffer[i].aBuffer[Index[i]][j:=j+1]:=DINT_TO_STRING(i_safetyCheckVar[i].m_slaveDriverOutput[1].m_cmdCurrent);  gCSV_Buffer[i].aBuffer[1][j]:='cmdTorqueIOJ6';
	gCSV_Buffer[i].aBuffer[Index[i]][j:=j+1]:=DINT_TO_STRING(i_safetyCheckVar[i].m_slaveDriverOutput[2].m_cmdCurrent);  gCSV_Buffer[i].aBuffer[1][j]:='cmdTorqueIOJ7';
	gCSV_Buffer[i].aBuffer[Index[i]][j:=j+1]:=DINT_TO_STRING(i_safetyCheckVar[i].m_slaveDriverOutput[3].m_cmdCurrent);  gCSV_Buffer[i].aBuffer[1][j]:='cmdTorqueIOJ8';

	//target motor encoder IO
	gCSV_Buffer[i].aBuffer[Index[i]][j:=j+1]:=DINT_TO_STRING(i_safetyCheckVar[i].m_setupDriverOutput[3].m_cmdMotorEncoder);  gCSV_Buffer[i].aBuffer[1][j]:='cmdMotorEncIOJ3';
	gCSV_Buffer[i].aBuffer[Index[i]][j:=j+1]:=DINT_TO_STRING(i_safetyCheckVar[i].m_setupDriverOutput[4].m_cmdMotorEncoder);  gCSV_Buffer[i].aBuffer[1][j]:='cmdMotorEncIOJ4';
	gCSV_Buffer[i].aBuffer[Index[i]][j:=j+1]:=DINT_TO_STRING(i_safetyCheckVar[i].m_setupDriverOutput[5].m_cmdMotorEncoder);  gCSV_Buffer[i].aBuffer[1][j]:='cmdMotorEncIOJ5';
	gCSV_Buffer[i].aBuffer[Index[i]][j:=j+1]:=DINT_TO_STRING(i_safetyCheckVar[i].m_slaveDriverOutput[1].m_cmdMotorEncoder);  gCSV_Buffer[i].aBuffer[1][j]:='cmdMotorEncIOJ6';
	gCSV_Buffer[i].aBuffer[Index[i]][j:=j+1]:=DINT_TO_STRING(i_safetyCheckVar[i].m_slaveDriverOutput[2].m_cmdMotorEncoder);  gCSV_Buffer[i].aBuffer[1][j]:='cmdMotorEncIOJ7';
	gCSV_Buffer[i].aBuffer[Index[i]][j:=j+1]:=DINT_TO_STRING(i_safetyCheckVar[i].m_slaveDriverOutput[3].m_cmdMotorEncoder);  gCSV_Buffer[i].aBuffer[1][j]:='cmdMotorEncIOJ8';


	//output motor opMode IO
	gCSV_Buffer[i].aBuffer[Index[i]][j:=j+1]:=DINT_TO_STRING(i_safetyCheckVar[i].m_setupDriverOutput[3].m_opMode);  gCSV_Buffer[i].aBuffer[1][j]:='opModeIOJ3';
	gCSV_Buffer[i].aBuffer[Index[i]][j:=j+1]:=DINT_TO_STRING(i_safetyCheckVar[i].m_setupDriverOutput[4].m_opMode);  gCSV_Buffer[i].aBuffer[1][j]:='opModeIOJ4';
	gCSV_Buffer[i].aBuffer[Index[i]][j:=j+1]:=DINT_TO_STRING(i_safetyCheckVar[i].m_setupDriverOutput[5].m_opMode);  gCSV_Buffer[i].aBuffer[1][j]:='opModeIOJ5';
	gCSV_Buffer[i].aBuffer[Index[i]][j:=j+1]:=DINT_TO_STRING(i_safetyCheckVar[i].m_slaveDriverOutput[1].m_opMode);  gCSV_Buffer[i].aBuffer[1][j]:='opModeIOJ6';
	gCSV_Buffer[i].aBuffer[Index[i]][j:=j+1]:=DINT_TO_STRING(i_safetyCheckVar[i].m_slaveDriverOutput[2].m_opMode);  gCSV_Buffer[i].aBuffer[1][j]:='opModeIOJ7';
	gCSV_Buffer[i].aBuffer[Index[i]][j:=j+1]:=DINT_TO_STRING(i_safetyCheckVar[i].m_slaveDriverOutput[3].m_opMode);  gCSV_Buffer[i].aBuffer[1][j]:='opModeIOJ8';


	END_IF
END_FOR
END_METHOD

METHOD cartDataCast : BOOL
VAR_IN_OUT CONSTANT
	i_safetyCheckVar : checkInputVariable;
	i_cartStatus : ST_CartStatus;
	i_cartJointData : ST_CartJointData;
END_VAR


IF ErrWritingFalg[5] = FALSE THEN
	c:=1;
	gCSV_Buffer[5].aBuffer[Index[5]][c:=c+1]:=LREAL_TO_FMTSTR(i_cartStatus.m_CartState,0, TRUE);  gCSV_Buffer[5].aBuffer[1][c]:='cartMachine';
	
	//cart Joint link position
	gCSV_Buffer[5].aBuffer[Index[5]][c:=c+1]:=LREAL_TO_STRING(i_cartJointData.m_curLinkPos[5]);  gCSV_Buffer[5].aBuffer[1][c]:='cartCurLinkPosJ5';
	gCSV_Buffer[5].aBuffer[Index[5]][c:=c+1]:=LREAL_TO_STRING(i_cartJointData.m_curLinkPos[6]);  gCSV_Buffer[5].aBuffer[1][c]:='cartCurLinkPosJ6';
	gCSV_Buffer[5].aBuffer[Index[5]][c:=c+1]:=LREAL_TO_STRING(i_cartJointData.m_curLinkPos[7]);  gCSV_Buffer[5].aBuffer[1][c]:='cartCurLinkPosJ7';
	gCSV_Buffer[5].aBuffer[Index[5]][c:=c+1]:=LREAL_TO_STRING(i_cartJointData.m_curLinkPos[8]);  gCSV_Buffer[5].aBuffer[1][c]:='cartCurLinkPosJ8';

	//cart current joint postion
	gCSV_Buffer[5].aBuffer[Index[5]][c:=c+1]:=LREAL_TO_STRING(i_cartJointData.m_curJntPos[5]);  gCSV_Buffer[5].aBuffer[1][c]:='curJntPosJ5';
	gCSV_Buffer[5].aBuffer[Index[5]][c:=c+1]:=LREAL_TO_STRING(i_cartJointData.m_curJntPos[6]);  gCSV_Buffer[5].aBuffer[1][c]:='curJntPosJ6';
	gCSV_Buffer[5].aBuffer[Index[5]][c:=c+1]:=LREAL_TO_STRING(i_cartJointData.m_curJntPos[7]);  gCSV_Buffer[5].aBuffer[1][c]:='curJntPosJ7';
	gCSV_Buffer[5].aBuffer[Index[5]][c:=c+1]:=LREAL_TO_STRING(i_cartJointData.m_curJntPos[8]);  gCSV_Buffer[5].aBuffer[1][c]:='curJntPosJ8';
	
	//cart target joint postion
	gCSV_Buffer[5].aBuffer[Index[5]][c:=c+1]:=LREAL_TO_STRING(i_cartJointData.m_cmdJntPos[5]);  gCSV_Buffer[5].aBuffer[1][c]:='cmdJntPosJ5';
	gCSV_Buffer[5].aBuffer[Index[5]][c:=c+1]:=LREAL_TO_STRING(i_cartJointData.m_cmdJntPos[6]);  gCSV_Buffer[5].aBuffer[1][c]:='cmdJntPosJ6';
	gCSV_Buffer[5].aBuffer[Index[5]][c:=c+1]:=LREAL_TO_STRING(i_cartJointData.m_cmdJntPos[7]);  gCSV_Buffer[5].aBuffer[1][c]:='cmdJntPosJ7';
	gCSV_Buffer[5].aBuffer[Index[5]][c:=c+1]:=LREAL_TO_STRING(i_cartJointData.m_cmdJntPos[8]);  gCSV_Buffer[5].aBuffer[1][c]:='cmdJntPosJ8';
	
	//drive error word
	gCSV_Buffer[5].aBuffer[Index[5]][c:=c+1]:=LREAL_TO_STRING(i_safetyCheckVar.m_cartDriverInput[1].m_driverError);  gCSV_Buffer[5].aBuffer[1][c]:='driverErrorJ1';
	gCSV_Buffer[5].aBuffer[Index[5]][c:=c+1]:=LREAL_TO_STRING(i_safetyCheckVar.m_cartDriverInput[2].m_driverError);  gCSV_Buffer[5].aBuffer[1][c]:='driverErrorJ2';
	gCSV_Buffer[5].aBuffer[Index[5]][c:=c+1]:=LREAL_TO_STRING(i_safetyCheckVar.m_cartDriverInput[6].m_driverError);  gCSV_Buffer[5].aBuffer[1][c]:='driverErrorJ6';
	gCSV_Buffer[5].aBuffer[Index[5]][c:=c+1]:=LREAL_TO_STRING(i_safetyCheckVar.m_cartDriverInput[7].m_driverError);  gCSV_Buffer[5].aBuffer[1][c]:='driverErrorJ7';
	gCSV_Buffer[5].aBuffer[Index[5]][c:=c+1]:=LREAL_TO_STRING(i_safetyCheckVar.m_cartDriverInput[8].m_driverError);  gCSV_Buffer[5].aBuffer[1][c]:='driverErrorJ8';
	
	//cart link encoder
	gCSV_Buffer[5].aBuffer[Index[5]][c:=c+1]:=LREAL_TO_STRING(i_safetyCheckVar.m_cartDriverInput[5].m_linkEncoder);  gCSV_Buffer[5].aBuffer[1][c]:='cartLinkIOJ5';
	gCSV_Buffer[5].aBuffer[Index[5]][c:=c+1]:=LREAL_TO_STRING(i_safetyCheckVar.m_cartDriverInput[6].m_linkEncoder);  gCSV_Buffer[5].aBuffer[1][c]:='cartLinkIOJ6';
	gCSV_Buffer[5].aBuffer[Index[5]][c:=c+1]:=LREAL_TO_STRING(i_safetyCheckVar.m_cartDriverInput[7].m_linkEncoder);  gCSV_Buffer[5].aBuffer[1][c]:='cartLinkIOJ7';
	gCSV_Buffer[5].aBuffer[Index[5]][c:=c+1]:=LREAL_TO_STRING(i_safetyCheckVar.m_cartDriverInput[8].m_linkEncoder);  gCSV_Buffer[5].aBuffer[1][c]:='cartLinkIOJ8';
	
	//cart actual torque 
	gCSV_Buffer[5].aBuffer[Index[5]][c:=c+1]:=DINT_TO_STRING(i_safetyCheckVar.m_cartDriverInput[1].m_current);  gCSV_Buffer[5].aBuffer[1][c]:='cartCurrentIOJ1';
	gCSV_Buffer[5].aBuffer[Index[5]][c:=c+1]:=DINT_TO_STRING(i_safetyCheckVar.m_cartDriverInput[2].m_current);  gCSV_Buffer[5].aBuffer[1][c]:='cartCurrentIOJ2';
	gCSV_Buffer[5].aBuffer[Index[5]][c:=c+1]:=DINT_TO_STRING(i_safetyCheckVar.m_cartDriverInput[6].m_current);  gCSV_Buffer[5].aBuffer[1][c]:='cartCurrentIOJ6';
	gCSV_Buffer[5].aBuffer[Index[5]][c:=c+1]:=DINT_TO_STRING(i_safetyCheckVar.m_cartDriverInput[7].m_current);  gCSV_Buffer[5].aBuffer[1][c]:='cartCurrentIOJ7';
	gCSV_Buffer[5].aBuffer[Index[5]][c:=c+1]:=DINT_TO_STRING(i_safetyCheckVar.m_cartDriverInput[8].m_current);  gCSV_Buffer[5].aBuffer[1][c]:='cartCurrentIOJ8';
	
	//cart joint status word
	gCSV_Buffer[5].aBuffer[Index[5]][c:=c+1]:=DINT_TO_STRING(i_safetyCheckVar.m_cartDriverInput[1].m_statusWord);  gCSV_Buffer[5].aBuffer[1][c]:='cartStatusWordIOJ1';
	gCSV_Buffer[5].aBuffer[Index[5]][c:=c+1]:=DINT_TO_STRING(i_safetyCheckVar.m_cartDriverInput[2].m_statusWord);  gCSV_Buffer[5].aBuffer[1][c]:='cartStatusWordIOJ2';
	gCSV_Buffer[5].aBuffer[Index[5]][c:=c+1]:=DINT_TO_STRING(i_safetyCheckVar.m_cartDriverInput[3].m_statusWord);  gCSV_Buffer[5].aBuffer[1][c]:='cartStatusWordIOJ3';
	gCSV_Buffer[5].aBuffer[Index[5]][c:=c+1]:=DINT_TO_STRING(i_safetyCheckVar.m_cartDriverInput[4].m_statusWord);  gCSV_Buffer[5].aBuffer[1][c]:='cartStatusWordIOJ4';
	gCSV_Buffer[5].aBuffer[Index[5]][c:=c+1]:=DINT_TO_STRING(i_safetyCheckVar.m_cartDriverInput[5].m_statusWord);  gCSV_Buffer[5].aBuffer[1][c]:='cartStatusWordIOJ5';
	gCSV_Buffer[5].aBuffer[Index[5]][c:=c+1]:=DINT_TO_STRING(i_safetyCheckVar.m_cartDriverInput[6].m_statusWord);  gCSV_Buffer[5].aBuffer[1][c]:='cartStatusWordIOJ6';
	gCSV_Buffer[5].aBuffer[Index[5]][c:=c+1]:=DINT_TO_STRING(i_safetyCheckVar.m_cartDriverInput[7].m_statusWord);  gCSV_Buffer[5].aBuffer[1][c]:='cartStatusWordIOJ7';
	gCSV_Buffer[5].aBuffer[Index[5]][c:=c+1]:=DINT_TO_STRING(i_safetyCheckVar.m_cartDriverInput[8].m_statusWord);  gCSV_Buffer[5].aBuffer[1][c]:='cartStatusWordIOJ8';
	
	//cart current joint motor encoder
	gCSV_Buffer[5].aBuffer[Index[5]][c:=c+1]:=DINT_TO_STRING(i_safetyCheckVar.m_cartDriverInput[1].m_motorEncoder);  gCSV_Buffer[5].aBuffer[1][c]:='cartCurMotorEncIOJ1';
	gCSV_Buffer[5].aBuffer[Index[5]][c:=c+1]:=DINT_TO_STRING(i_safetyCheckVar.m_cartDriverInput[2].m_motorEncoder);  gCSV_Buffer[5].aBuffer[1][c]:='cartCurMotorEncIOJ2';
	gCSV_Buffer[5].aBuffer[Index[5]][c:=c+1]:=DINT_TO_STRING(i_safetyCheckVar.m_cartDriverInput[3].m_motorEncoder);  gCSV_Buffer[5].aBuffer[1][c]:='cartCurMotorEncIOJ3';
	gCSV_Buffer[5].aBuffer[Index[5]][c:=c+1]:=DINT_TO_STRING(i_safetyCheckVar.m_cartDriverInput[4].m_motorEncoder);  gCSV_Buffer[5].aBuffer[1][c]:='cartCurMotorEncIOJ4';
	gCSV_Buffer[5].aBuffer[Index[5]][c:=c+1]:=DINT_TO_STRING(i_safetyCheckVar.m_cartDriverInput[5].m_motorEncoder);  gCSV_Buffer[5].aBuffer[1][c]:='cartCurMotorEncIOJ5';
	gCSV_Buffer[5].aBuffer[Index[5]][c:=c+1]:=DINT_TO_STRING(i_safetyCheckVar.m_cartDriverInput[6].m_motorEncoder);  gCSV_Buffer[5].aBuffer[1][c]:='cartCurMotorEncIOJ6';
	gCSV_Buffer[5].aBuffer[Index[5]][c:=c+1]:=DINT_TO_STRING(i_safetyCheckVar.m_cartDriverInput[7].m_motorEncoder);  gCSV_Buffer[5].aBuffer[1][c]:='cartCurMotorEncIOJ7';
	gCSV_Buffer[5].aBuffer[Index[5]][c:=c+1]:=DINT_TO_STRING(i_safetyCheckVar.m_cartDriverInput[8].m_motorEncoder);  gCSV_Buffer[5].aBuffer[1][c]:='cartCurMotorEncIOJ8';

	//cart commend joint motor encoder
	gCSV_Buffer[5].aBuffer[Index[5]][c:=c+1]:=DINT_TO_STRING(i_safetyCheckVar.m_cartDriverOutput[1].m_cmdMotorEncoder);  gCSV_Buffer[5].aBuffer[1][c]:='cartCmdMotorEncIOJ1';
	gCSV_Buffer[5].aBuffer[Index[5]][c:=c+1]:=DINT_TO_STRING(i_safetyCheckVar.m_cartDriverOutput[2].m_cmdMotorEncoder);  gCSV_Buffer[5].aBuffer[1][c]:='cartCmdMotorEncIOJ2';
	gCSV_Buffer[5].aBuffer[Index[5]][c:=c+1]:=DINT_TO_STRING(i_safetyCheckVar.m_cartDriverOutput[3].m_cmdMotorEncoder);  gCSV_Buffer[5].aBuffer[1][c]:='cartCmdMotorEncIOJ3';
	gCSV_Buffer[5].aBuffer[Index[5]][c:=c+1]:=DINT_TO_STRING(i_safetyCheckVar.m_cartDriverOutput[4].m_cmdMotorEncoder);  gCSV_Buffer[5].aBuffer[1][c]:='cartCmdMotorEncIOJ4';
	gCSV_Buffer[5].aBuffer[Index[5]][c:=c+1]:=DINT_TO_STRING(i_safetyCheckVar.m_cartDriverOutput[5].m_cmdMotorEncoder);  gCSV_Buffer[5].aBuffer[1][c]:='cartCmdMotorEncIOJ5';
	gCSV_Buffer[5].aBuffer[Index[5]][c:=c+1]:=DINT_TO_STRING(i_safetyCheckVar.m_cartDriverOutput[6].m_cmdMotorEncoder);  gCSV_Buffer[5].aBuffer[1][c]:='cartCmdMotorEncIOJ6';
	gCSV_Buffer[5].aBuffer[Index[5]][c:=c+1]:=DINT_TO_STRING(i_safetyCheckVar.m_cartDriverOutput[7].m_cmdMotorEncoder);  gCSV_Buffer[5].aBuffer[1][c]:='cartCmdMotorEncIOJ7';
	gCSV_Buffer[5].aBuffer[Index[5]][c:=c+1]:=DINT_TO_STRING(i_safetyCheckVar.m_cartDriverOutput[8].m_cmdMotorEncoder);  gCSV_Buffer[5].aBuffer[1][c]:='cartCmdMotorEncIOJ8';	
END_IF
END_METHOD

METHOD errCodeAnalysis : BOOL
VAR_INPUT
END_VAR

FOR i:=1 TO g_maxNum BY 1 DO
	IF g_ArrayErrCodeArm[i][0]<>0 AND ArrayErrCodeTypeLast[i]<> g_ArrayErrCodeArm[i][0]  THEN
		arm:=SHR(g_ArrayErrCodeArm[i][0],24)-3;
		IF arm>g_maxNum THEN
			arm:=g_maxNum;	
		END_IF
		Joint:=SHR(g_arrayErrCodeArm[i][0],16) AND 16#FF;
		ErrID:=g_arrayErrCodeArm[i][0];
		mErrNameLocation[arm,1]:=LREAL_TO_FMTSTR(Arm,0, TRUE);
		mErrNameLocation[arm,2]:=LREAL_TO_FMTSTR(Joint,0, TRUE);
		mErrNameLocation[arm,3]:=DWORD_TO_HEXSTR(UDINT_TO_DWORD(ErrID),0, TRUE);
		m_Index[arm]:=INT_TO_UDINT(Index[arm]);
		errWritingAllowed[arm]:=TRUE;
	END_IF
	ArrayErrCodeTypeLast[i]:=g_ArrayErrCodeArm[i][0];
	errFlagDelay1s[i](IN:= errWritingAllowed[i], PT:= T#2S, Q=> errWritingFalg[i], ET=> );
END_FOR
END_METHOD

METHOD run : BOOL
VAR_IN_OUT CONSTANT
	i_safetyCheckVar :ARRAY[1..g_maxNum] OF checkInputVariable;
	i_cartStatus : ST_CartStatus;
	i_cartJointData : ST_CartJointData;
	i_setupStatus : ST_SetupStatus;
	i_slaveStatus : ST_SlaveStatus;
	i_setupJointData : ST_SetupJointData;
	i_slaveJointData : ST_SlaveJointData;
END_VAR
_tNow := systemTime();
IF _tNow.wYear = 0 THEN
	RETURN;
END_IF

errCodeAnalysis();

armDataCast(i_safetyCheckVar,i_setupStatus,i_slaveStatus,i_setupJointData,i_slaveJointData);

cartDataCast(i_safetyCheckVar[5],i_cartStatus,i_cartJointData);

FOR _iBuffer := 1 TO MAX_CSV_RING_BUFFER BY 1 DO
	TransferToWrittenVariable();

	WriterCSV();
	
	StartRecord[_iBuffer](CLK:=ErrWritingFalg[_iBuffer] , Q=> );

	IF ErrWritingFalg[_iBuffer] =FALSE THEN
		Index[_iBuffer]:=Index[_iBuffer]+1;
		IF Index[_iBuffer]>10000 THEN
			index[_iBuffer]:=2;
		END_IF
	END_IF
	
END_FOR
END_METHOD

METHOD systemTime : TIMESTRUCT
VAR_INPUT
END_VAR
fbSysTime(timeLoDW=>tFileTime.dwLowDateTime , timeHiDW=> tFileTime.dwHighDateTime);

_tNowBoLin := FILETIME_TO_SYSTEMTIME(tFileTime);
systemTime:=_tNowBoLin;
systemTime.wHour:=_tNowBoLin.wHour+8;
IF systemTime.wHour>23 THEN
	systemTime.wHour:=_tNow.wHour-24;
END_IF
END_METHOD

METHOD TransferToWrittenVariable : BOOL
VAR_INPUT
END_VAR
	

	gCSV_Buffer[_iBuffer].aBuffer[Index[_iBuffer]][0]:= SYSTEMTIME_TO_STRING(_tNow);(*第二行第一列*)
	gCSV_Buffer[_iBuffer].aBuffer[Index[_iBuffer]][1]:=LREAL_TO_FMTSTR(Index[_iBuffer],0, TRUE); 
	
	(*The first line shows the arm joint and the error name*)
	mErrNameLocation[_iBuffer,0] := INT_TO_STRING(Index[_iBuffer]);
	gCSV_Buffer[_iBuffer].aBuffer[0][0] := mErrNameLocation[_iBuffer,0];
	gCSV_Buffer[_iBuffer].aBuffer[0][1] := mErrNameLocation[_iBuffer,1];
	gCSV_Buffer[_iBuffer].aBuffer[0][2] := mErrNameLocation[_iBuffer,2];
	gCSV_Buffer[_iBuffer].aBuffer[0][3] := mErrNameLocation[_iBuffer,3];
	//gCSV_Buffer[_iBuffer].aBuffer[4][0] := mErrNameLocation[_iBuffer,4];
	
	(*The second line shows the variable name*)
	gCSV_Buffer[_iBuffer].aBuffer[1][0] := 'SystemTime';
	gCSV_Buffer[_iBuffer].aBuffer[1][1] := 'Index';

	sPath:= 'C:\Robot\Error\'; 
	mErr[0]:=CONCAT('Arm',mErrNameLocation[_iBuffer,1]);
	mErr[1]:=CONCAT('Joint',mErrNameLocation[_iBuffer,2]);
	mErr[2]:=mErrNameLocation[_iBuffer,3];
	IF StartRecord[_iBuffer].Q THEN  
	gCSV_Buffer[_iBuffer].bFull := TRUE;
	fbFormat( 	sFormat := _sPathFormat ,
			 	arg1 := F_STRING(sPath),   arg2 := F_WORD(_tNow.wYear), arg3 := F_WORD(_tNow.wMonth), 
				arg4 := F_WORD(_tNow.wDay), arg5 := F_WORD(_tNow.wHour),arg6 := F_WORD(_tNow.wMinute),arg7 := F_WORD(_tNow.wSecond),
			    arg8 := F_STRING(mErr[0]),arg9 := F_STRING(mErr[1]),arg10 := F_STRING(mErr[2]),  sOut => gCSV_Buffer[_iBuffer].sPath);
	END_IF

	//F_STRING(mErr[0])
END_METHOD

METHOD writerCSV : BOOL
VAR_INPUT
END_VAR

IF gCSV_Buffer[_iBuffer].bFull THEN
	gCSV_Buffer[_iBuffer].fbWriter(bWrite:= gCSV_Buffer[_iBuffer].bFull,sFileName:=gCSV_Buffer[_iBuffer].sPath, pBuffer :=ADR(gCSV_Buffer[_iBuffer].aBuffer),Index:=m_Index[_iBuffer]);
	gCSV_Buffer[_iBuffer].bFull := gCSV_Buffer[_iBuffer].fbWriter.bBusy;
END_IF


RecordCompletion[_iBuffer](CLK:= gCSV_Buffer[_iBuffer].bFull, Q=> );
IF RecordCompletion[_iBuffer].Q THEN
	errWritingAllowed[_iBuffer]:=FALSE;
	Index[_iBuffer]:=2;
	gCSV_Buffer[_iBuffer].aBuffer:=iZeroRowsData;
	g_ArrayErrCodeArm[_iBuffer]:=iZeroErrCode[_iBuffer];
	//gCSV_Buffer[_iBuffer].fbWriter.arrDataForward(array_in:=Robot_Status.ArrayErrCodeType[_iBuffer]  , array_out=> Robot_Status.ArrayErrCodeType[_iBuffer]);
END_IF
END_METHOD

END_FUNCTION_BLOCK

// ---- FBs_CartControlles/FB_CartCtrlError.TcPOU
FUNCTION_BLOCK FB_CartCtrlError EXTENDS FB_CartCtrlBase
VAR_INPUT
END_VAR
VAR_OUTPUT
END_VAR
VAR
END_VAR

// override this function in each exact controller
METHOD PROTECTED calcCmdJntPos : BOOL
VAR_IN_OUT CONSTANT
	// slave cart joint data
	i_slaveCart :FB_SlaveCart;
END_VAR
m_cmdJntPos := i_slaveCart.curJntPos;
END_METHOD

// override this function in each exact controller
// NOTICE: set joint control mode here, and do some initialization if needed
METHOD PUBLIC init : BOOL
VAR_IN_OUT CONSTANT
	i_slaveCart	:FB_SlaveCart;
END_VAR
VAR_IN_OUT 
	r_cartCtrlCmd :ST_SlaveArmCtrlCmds;
END_VAR
SUPER^.init(i_slaveCart,r_cartCtrlCmd);

// update commands to arm
copyCmds(r_cartCtrlCmd);
END_METHOD

END_FUNCTION_BLOCK

// ---- FBs_CartControlles/FB_CartCtrlBase.TcPOU
// Slave Arm Base Controller, Hold at Current Posture
FUNCTION_BLOCK FB_CartCtrlBase IMPLEMENTS I_CartJointCtrl
VAR_INPUT
END_VAR
VAR_OUTPUT
END_VAR
VAR
	// flag if the controller has finished all its jobs
	m_isFinished:BOOL:=FALSE;
	
	// controller execute time period
	m_timePeriod :LREAL:=0;
	
	// flag to hold last commands
	m_holdLastCmds :BOOL := FALSE;
	
	// arm control data
	// NOTE: simulated joint position is usd for kinematic controller 
	//		while command joint position is used for real robot controller
	// 		They are identical for the most time, but in some cases, simulated position is filted to get command one 
	m_cmdJntPos : VEC8d; 
	m_cmdJntVel : VEC8d;
	m_cmdJntAcc : VEC8d;
	m_cmdJntTrq : VEC8d;
	m_jntOPMode : Vec8i;
	m_jntEnableFlag :Vec8i;

	
END_VAR

// override this function in each exact controller
METHOD PROTECTED calcCmdJntPos : BOOL
VAR_IN_OUT CONSTANT
	// slave cart joint data
	i_slaveCart :FB_SlaveCart;
END_VAR
IF isFinished THEN
	RETURN;
END_IF
END_METHOD

// override this function in each exact controller
METHOD PROTECTED calcCmdJntVel : BOOL
VAR_IN_OUT CONSTANT
	// slave cart joint data
	i_slaveCart :FB_SlaveCart;
END_VAR
IF isFinished THEN
	RETURN;
END_IF

// set joint torque to zero in default
//m_cmdJntVel := g_zeroVec8d;
END_METHOD

METHOD checkToHoldLastCmds : BOOL
VAR_IN_OUT CONSTANT
	// slave cart joint data
	i_slaveCart :FB_SlaveCart;
END_VAR
VAR
	j:INT;
	maxJntErr:LREAL;
	jntCtrlErr:Vec8d;
END_VAR
// check if to hold the command joint position unchanged
vecSub(i_slaveCart.m_cmdJntPos, i_slaveCart.m_curJntPos,jntCtrlErr);
maxJntErr:=0.0;
FOR j:=1 TO g_cartJntNum DO
	maxJntErr:= MAX(maxJntErr, ABS(jntCtrlErr[j]));
END_FOR

checkToHoldLastCmds := (maxJntErr<GVL_SlaveControlParameters.g_jntCtrlErrForCmdHold);
END_METHOD

METHOD copyCmds : BOOL
VAR_IN_OUT 
	r_cartCtrlCmd :ST_SlaveArmCtrlCmds;
END_VAR
r_cartCtrlCmd.m_jntEnableFlag :=m_jntEnableFlag;
r_cartCtrlCmd.m_cmdJntPos:=m_cmdJntPos;
r_cartCtrlCmd.m_cmdJntVel:=m_cmdJntVel;
r_cartCtrlCmd.m_cmdJntAcc:=m_cmdJntAcc;
r_cartCtrlCmd.m_cmdJntTrq:=m_cmdJntTrq;
r_cartCtrlCmd.m_jntOPMode:=m_jntOPMode;
END_METHOD

// override this function in each exact controller
// NOTICE: set joint control mode here, and do some initialization if needed
METHOD PUBLIC init : BOOL
VAR_IN_OUT CONSTANT
	// slave cart joint data
	i_slaveCart :FB_SlaveCart;
END_VAR
VAR_IN_OUT 
	r_cartCtrlCmd :ST_SlaveArmCtrlCmds;
END_VAR
m_timePeriod:=0;
m_jntEnableFlag :=g_zeroVec8i;
m_jntOPMode:=g_slaveAllPosMode;

IF FALSE = m_holdLastCmds THEN
	m_cmdJntPos:=i_slaveCart.m_curJntPos;
ELSE
	m_cmdJntPos:=r_cartCtrlCmd.m_cmdJntPos;
END_IF

m_cmdJntVel:=g_zeroVec8d;
m_cmdJntAcc:=g_zeroVec8d;
m_cmdJntTrq:=g_zeroVec8d;

// update commands to arm
copyCmds(r_cartCtrlCmd);
END_METHOD

PROPERTY isFinished : BOOL
GET
isFinished:=m_isFinished;
END_GET
END_PROPERTY

{warning '添加方法实现'}
METHOD reset : BOOL
m_isFinished:=FALSE;
m_timePeriod:=0;
END_METHOD

{warning '添加方法实现'}
METHOD run : BOOL
VAR_IN_OUT CONSTANT
	// slave cart joint data
	i_slaveCart :FB_SlaveCart;
END_VAR
VAR_IN_OUT
	r_cartCtrlCmd :ST_SlaveArmCtrlCmds;
END_VAR
VAR
	i:INT;
END_VAR
IF m_isFinished THEN
	RETURN;
END_IF

// check if arm enabled
//IF FALSE = i_slaveCartJoint.isEnabled(m_jntEnableFlag) THEN
//	RETURN;
//END_IF

// calculate command joint position--Motion control
calcCmdJntPos( i_slaveCart);

// calculate command joint torque -- Force control
calcCmdJntVel(i_slaveCart);

// update commands to arm
copyCmds(r_cartCtrlCmd);

// update time period
m_timePeriod := m_timePeriod+g_slaveArmCtrlCycleTime;
END_METHOD

END_FUNCTION_BLOCK

// ---- FBs_CartControlles/FB_CartCtrlInit.TcPOU
FUNCTION_BLOCK FB_CartCtrlInit EXTENDS FB_CartCtrlBase
VAR_INPUT
END_VAR
VAR_OUTPUT
END_VAR
VAR
END_VAR

// override this function in each exact controller
METHOD PROTECTED calcCmdJntPos : BOOL
VAR_IN_OUT CONSTANT
	// slave cart joint data
	i_slaveCart :FB_SlaveCart;
END_VAR
IF m_timePeriod > 1.0 THEN
	m_isFinished := true;
END_IF
END_METHOD

// override this function in each exact controller
// NOTICE: set joint control mode here, and do some initialization if needed
METHOD PUBLIC init : BOOL
VAR_IN_OUT CONSTANT
	i_slaveCart	:FB_SlaveCart;
END_VAR
VAR_IN_OUT 
	r_cartCtrlCmd :ST_SlaveArmCtrlCmds;
END_VAR
SUPER^.init(i_slaveCart,r_cartCtrlCmd);

// update commands to arm
copyCmds(r_cartCtrlCmd);
END_METHOD

END_FUNCTION_BLOCK

// ---- FBs_CartControlles/FB_CartCtrlReady.TcPOU
FUNCTION_BLOCK FB_CartCtrlReady EXTENDS FB_CartCtrlBase
VAR_INPUT
END_VAR
VAR_OUTPUT
END_VAR
VAR
END_VAR

// override this function in each exact controller
METHOD PROTECTED calcCmdJntPos : BOOL
VAR_IN_OUT CONSTANT
	// slave cart joint data
	i_slaveCart :FB_SlaveCart;
END_VAR
//m_cmdJntPos := i_slaveCart.curJntPos;
END_METHOD

// override this function in each exact controller
// NOTICE: set joint control mode here, and do some initialization if needed
METHOD PUBLIC init : BOOL
VAR_IN_OUT CONSTANT
	i_slaveCart	:FB_SlaveCart;
END_VAR
VAR_IN_OUT 
	r_cartCtrlCmd :ST_SlaveArmCtrlCmds;
END_VAR
//m_holdLastCmds := checkToHoldLastCmds(i_slaveCart);
m_holdLastCmds := checkToHoldLastCmds(i_slaveCart);
SUPER^.init(i_slaveCart,r_cartCtrlCmd);

// update commands to arm
copyCmds(r_cartCtrlCmd);
END_METHOD

END_FUNCTION_BLOCK

// ---- FBs_CartControlles/FB_CartCtrlInSurgery.TcPOU
FUNCTION_BLOCK FB_CartCtrlInSurgery EXTENDS FB_CartCtrlBase
VAR_INPUT
END_VAR
VAR_OUTPUT
END_VAR
VAR
END_VAR

// override this function in each exact controller
METHOD PROTECTED calcCmdJntPos : BOOL
VAR_IN_OUT CONSTANT
	// slave cart joint data
	i_slaveCart :FB_SlaveCart;
END_VAR
m_cmdJntPos := i_slaveCart.curJntPos;
END_METHOD

// override this function in each exact controller
// NOTICE: set joint control mode here, and do some initialization if needed
METHOD PUBLIC init : BOOL
VAR_IN_OUT CONSTANT
	i_slaveCart	:FB_SlaveCart;
END_VAR
VAR_IN_OUT 
	r_cartCtrlCmd :ST_SlaveArmCtrlCmds;
END_VAR
//m_holdLastCmds := checkToHoldLastCmds(i_slaveCart);
m_holdLastCmds := checkToHoldLastCmds(i_slaveCart);
SUPER^.init(i_slaveCart,r_cartCtrlCmd);

// update commands to arm
copyCmds(r_cartCtrlCmd);
END_METHOD

END_FUNCTION_BLOCK

// ---- FBs_CartControlles/FB_CartCtrlMotionCar.TcPOU
FUNCTION_BLOCK FB_CartCtrlMotionCar EXTENDS FB_CartCtrlBase
VAR_INPUT
END_VAR
VAR_OUTPUT
END_VAR
VAR
	m_driveForce: ARRAY [1..2] OF LREAL;
	
	// input drive force filter
	m_driveVelLpf : ARRAY [1..2] OF FB_LowPassFilter;
	m_driveForceFilter: Vec2i;
	
	//cart motion trajectory velocity
	m_trajVel : ARRAY [1..2] OF LREAL;
	m_motorDir :ARRAY [1..2] OF INT := [1,-1];
	
	m_tarJntPos : ARRAY [1..2] OF LREAL;
	m_incJntPos : ARRAY [1..2] OF LREAL;
	m_initJntPos : ARRAY [1..2] OF LREAL;
	// time threshold to drive wheel after it's enabled
	m_cartWheelDriveWaitTime :LREAL := 0.2;
	
	//wheel motion  time 
	m_wheelMotionTime:ARRAY [1..2] OF LREAL;
	
	// filter cut-off frequency for cart drive force 
	m_cmdJntVelLpfCutoffFreq : LREAL :=5;
END_VAR

VAR CONSTANT
	//Proportionality constant of force sensor
	m_driveForceProConstant : LREAL := 5/15000;
END_VAR

// override this function in each exact controller
METHOD PROTECTED calcCmdJntPos : BOOL
VAR_IN_OUT CONSTANT
	// slave cart joint data
	i_slaveCart :FB_SlaveCart;
END_VAR

VAR
	i:INT;
END_VAR

FOR i := 1 TO 2 BY 1 DO
	m_driveForce[i] :=LIMIT(-5, i_slaveCart.m_driveForce[i]/3000, 5);
	m_wheelMotionTime[i] := LIMIT(0, m_wheelMotionTime[i] + g_cartCtrlCycleTime, 1);
	
	IF m_wheelMotionTime[i] > m_cartWheelDriveWaitTime THEN
		m_trajVel[i] := m_driveVelLpf[i].run(i_rawData:=m_motorDir[i] * m_driveForce[i]/2);
		m_incJntPos[i] := m_incJntPos[i] + m_trajVel[i] * g_cartCtrlCycleTime;
		
		m_cmdJntPos[i+2] := m_initJntPos[i] + m_incJntPos[i];
	END_IF
END_FOR
END_METHOD

// override this function in each exact controller
// NOTICE: set joint control mode here, and do some initialization if needed
METHOD PUBLIC init : BOOL
VAR_IN_OUT CONSTANT
	i_slaveCart	:FB_SlaveCart;
END_VAR
VAR_IN_OUT 
	r_cartCtrlCmd :ST_SlaveArmCtrlCmds;
END_VAR
//m_holdLastCmds := checkToHoldLastCmds(i_slaveCart);
m_holdLastCmds := checkToHoldLastCmds(i_slaveCart);
SUPER^.init(i_slaveCart,r_cartCtrlCmd);

m_jntEnableFlag[3] :=1;
m_jntEnableFlag[4] :=1;

m_jntOPMode[3]:= DriverOPMode_cspMZ;
m_jntOPMode[4]:= DriverOPMode_cspMZ;

m_tarJntPos[1] := 0;
m_tarJntPos[2] := 0;

m_incJntPos[1] := 0;
m_incJntPos[2] := 0;

m_initJntPos[1] := i_slaveCart.curJntPos[3];
m_initJntPos[2] := i_slaveCart.curJntPos[4];

m_driveVelLpf[1].init(i_filterOrd:= 1, i_cutoffFreq:= m_cmdJntVelLpfCutoffFreq, i_sampleFreq:= 8000);
m_driveVelLpf[2].init(i_filterOrd:= 1, i_cutoffFreq:= m_cmdJntVelLpfCutoffFreq, i_sampleFreq:= 8000);

m_driveVelLpf[1].run(i_rawData:=0);
m_driveVelLpf[2].run(i_rawData:=0);


m_wheelMotionTime[1]:=0;
m_wheelMotionTime[2]:=0;

// update commands to arm
copyCmds(r_cartCtrlCmd);
END_METHOD

END_FUNCTION_BLOCK

// ---- FBs_CartControlles/FB_CartCtrlAsepticDeploy.TcPOU
FUNCTION_BLOCK FB_CartCtrlAsepticDeploy EXTENDS FB_CartCtrlBase
VAR_INPUT
END_VAR
VAR_OUTPUT
END_VAR
VAR

	m_actJntPos: Vec8d;
	m_tarJntPos: Vec8d;
	m_jntPosArrival : Vec8b;
	m_initActJntPos: Vec8d;
	m_initTarJntPos : Vec8d;
	m_incTarJntPos : Vec8d;

	// time threshold to 5-8joint after it's enabled
	m_cartAdjustStartWaitTime :LREAL := 0.3;
	
	//adjust start  time 
	m_adjustStartTime :LREAL;
	
	m_jntOTG :ARRAY[1..8] OF FB_secOrdTrajFilter;
	//m_trajPlan :ARRAY[1..8] OF TrapezoIDal_velocity_trajectory;
END_VAR

// override this function in each exact controller
METHOD PROTECTED calcCmdJntPos : BOOL
VAR_IN_OUT CONSTANT
	// slave cart joint data
	i_slaveCart :FB_SlaveCart;
END_VAR

VAR
	i:INT;
	actPosErr : vec8d;
	tarPosErr : vec8d;
END_VAR
//In this method, 5 represents the pillar postion , 6 represents the beam rotation angle ,7 represents the beam stretch position ,8 represents the overhang angle
m_adjustStartTime :=LIMIT(0, m_adjustStartTime + g_cartCtrlCycleTime, 1);
m_actJntPos := i_slaveCart.curJntPos;
IF i_slaveCart.ctrlEnable.m_dockingEnable THEN
	m_initTarJntPos := i_slaveCart.m_cartDataFromUI.m_cartSpecificPosDocking;
ELSIF i_slaveCart.ctrlEnable.m_drapingEnable THEN
	m_initTarJntPos := i_slaveCart.m_cartDataFromUI.m_cartSpecificPosDraping;
END_IF
vecSub(m_initTarJntPos, m_actJntPos, actPosErr);
vecSub(m_initTarJntPos, m_tarJntPos, tarPosErr);

IF m_adjustStartTime >= m_cartAdjustStartWaitTime THEN
	FOR i := 5 TO 8 BY 1 DO
		IF ABS(actPosErr[i]) <= GVL_CartControlParameters.g_jntCtrlAngTolHigh*2  THEN
			m_jntPosArrival[i] := TRUE;
		END_IF
		
		IF ABS(tarPosErr[i]) > GVL_CartControlParameters.g_jntCtrlAngTolHigh THEN
			m_incTarJntPos[i] := m_incTarJntPos[i] + sign(actPosErr[i]) * GVL_CartControlParameters.g_maxJntVel[i]/2 * g_cartCtrlCycleTime;
			m_tarJntPos[i] := m_actJntPos[i] + m_incTarJntPos[i];
		END_IF
	END_FOR
	
	IF m_jntPosArrival[5] AND m_jntPosArrival[6] AND m_jntPosArrival[7] AND m_jntPosArrival[8] THEN
		m_isFinished := TRUE;
	END_IF
	
	FOR i := 5 TO 8 BY 1 DO
		m_jntOTG[i].run(i_targetPos:= m_tarJntPos[i], i_targetVel:= 0.0, o_cmdAcc=> , o_cmdVel=> , o_cmdPos=>m_cmdJntPos[i] );
	END_FOR
END_IF
END_METHOD

// override this function in each exact controller
// NOTICE: set joint control mode here, and do some initialization if needed
METHOD PUBLIC init : BOOL
VAR_IN_OUT CONSTANT
	i_slaveCart	:FB_SlaveCart;
END_VAR
VAR_IN_OUT 
	r_cartCtrlCmd :ST_SlaveArmCtrlCmds;
END_VAR
VAR
	i : INT;
END_VAR
m_holdLastCmds := checkToHoldLastCmds(i_slaveCart);
SUPER^.init(i_slaveCart,r_cartCtrlCmd);

m_jntEnableFlag[5] :=1;
m_jntEnableFlag[6] :=1;
m_jntEnableFlag[7] :=1;
m_jntEnableFlag[8] :=1;

m_jntOPMode[5]:= DriverOPMode_cspMZ;
m_jntOPMode[6]:= DriverOPMode_Pos;
m_jntOPMode[7]:= DriverOPMode_Pos;
m_jntOPMode[8]:= DriverOPMode_Pos;

m_initActJntPos:=m_cmdJntPos;//i_slaveCart.curJntPos;
m_jntPosArrival := g_zeroVec8b;
m_incTarJntPos := g_zeroVec8d;
m_tarJntPos := g_zeroVec8d;
m_jntPosArrival := g_zeroVec8b;

IF i_slaveCart.ctrlEnable.m_dockingEnable THEN
	m_initTarJntPos := i_slaveCart.m_cartDataFromUI.m_cartSpecificPosDocking;
ELSIF i_slaveCart.ctrlEnable.m_drapingEnable THEN
	m_initTarJntPos := i_slaveCart.m_cartDataFromUI.m_cartSpecificPosDraping;
END_IF

FOR i := 1 TO 4 BY 1 DO
	m_jntOTG[i+4].init(i_curCmdPos:= m_cmdJntPos[i+4], i_curCmdVel:= 0, i_maxV:=GVL_CartControlParameters.g_maxJntVel[i+4] , i_maxA:=GVL_CartControlParameters.g_maxJntAcc[i+4] , i_Ts:=g_cartCtrlCycleTime );
END_FOR
//m_initTarJntPos := m_tarJntPos;
m_adjustStartTime := 0;
// update commands to arm
copyCmds(r_cartCtrlCmd);
END_METHOD

END_FUNCTION_BLOCK

// ---- FBs_CartControlles/FB_CartCtrlAdjust.TcPOU
FUNCTION_BLOCK FB_CartCtrlAdjust EXTENDS FB_CartCtrlBase
VAR_INPUT
END_VAR
VAR_OUTPUT
END_VAR
VAR

	m_joystickSignal: Vec8d;	
	m_fiducialValue:INT:= 512;
	m_joystickRange:INT:=430;
	m_joystickDir: Vec8i:=[1,1,1,1,-1,-1,1,1];
	m_joystickVelInc: Vec8d;
	m_actJntPos: Vec8d;
	m_tarPosInc: Vec8d;
	m_lastPosInc: Vec8d;
	m_tarCartPos: Vec8d;
	m_trajJntPos : Vec8d;
	m_tarJntPos : Vec8d;
	m_initActJntPos: Vec8d;
	m_initActCartPos: Vec8d;
	m_veiwAngle : LREAL;
	m_jntPosReachLimit : Vec8b;
	m_maxJntPos : vec8d;

	m_carJntSoftwareLimit :ARRAY [5..8] OF LREAL := [0.005, 2*g_deg2Rad, 0.005, 2*g_deg2Rad];
	
	// time threshold to 5-8joint after it's enabled
	m_cartAdjustStartWaitTime :LREAL := 0.3;
	
	//adjust start  time 
	m_adjustStartTime :LREAL;
	
	// filter cut-off frequency for cart drive force 
	m_cmdJoystickLpfCutoffFreq : LREAL :=8;
	m_cartCtrlFreq :LREAL:=8000;
	
	m_jntOTG :ARRAY[1..8] OF FB_secOrdTrajFilter;
END_VAR

// override this function in each exact controller
METHOD PROTECTED calcCmdJntPos : BOOL
VAR_IN_OUT CONSTANT
	// slave cart joint data
	i_slaveCart :FB_SlaveCart;
END_VAR

VAR
	i:INT;
END_VAR
//In this method, 5 represents the pillar postion , 6 represents the beam rotation angle ,7 represents the beam stretch position ,8 represents the overhang angle
m_adjustStartTime :=LIMIT(0, m_adjustStartTime + g_cartCtrlCycleTime, 1);
m_actJntPos := i_slaveCart.curJntPos;
m_actJntPos[7] := i_slaveCart.curJntPos[7] + GVL_CartControlParameters.g_curBeamStretchJntInitPos;
m_veiwAngle := m_actJntPos[6] + m_actJntPos[8];

IF m_adjustStartTime > m_cartAdjustStartWaitTime THEN
	FOR i:= 1 TO 4 BY 1 DO
		m_joystickSignal[i] := i_slaveCart.m_joystickSignal[i] - m_fiducialValue;
		m_joystickVelInc[i+4] := m_joystickSignal[i]/m_joystickRange*m_joystickDir[i+4]*GVL_CartControlParameters.g_maxCartVel[i];
		m_tarPosInc[i+4] := m_tarPosInc[i+4] + m_joystickVelInc[i+4] * g_cartCtrlCycleTime;
	END_FOR
	
	m_tarCartPos[5] := m_initActJntPos[5] + m_tarPosInc[5];
	IF i_slaveCart.m_ctrlEnable.m_cameraJoystickEnable THEN
		m_tarCartPos[6] := m_initActCartPos[6] + m_tarPosInc[6]*COS(m_veiwAngle)+m_tarPosInc[7]*SIN(m_veiwAngle);
		m_tarCartPos[7] := m_initActCartPos[7] - m_tarPosInc[6]*SIN(m_veiwAngle)+m_tarPosInc[7]*COS(m_veiwAngle);
	ELSE
		m_tarCartPos[6] := m_initActCartPos[6] + m_tarPosInc[6];
		m_tarCartPos[7] := m_initActCartPos[7] + m_tarPosInc[7];
	END_IF
	m_tarCartPos[8] := m_initActJntPos[8] + m_tarPosInc[8];
	
	IF i_slaveCart.m_ctrlEnable.m_heightLimitAdjustEnable THEN
		m_trajJntPos[5] := m_tarCartPos[5];
	ELSE
		m_trajJntPos[5] := LIMIT(GVL_CartMotorParameters.g_minJntPos[5], m_tarCartPos[5], MAX(m_actJntPos[5],i_slaveCart.m_cartDataFromUI.m_standColumnHightLimit));
	END_IF
	m_trajJntPos[6] := atan2( m_tarCartPos[6], m_tarCartPos[7]);
	m_trajJntPos[7] := m_tarCartPos[7]/COS(m_trajJntPos[6]) - GVL_CartControlParameters.g_curBeamStretchJntInitPos;
	m_trajJntPos[8] := m_tarCartPos[8] -  (m_trajJntPos[6] - m_initActJntPos[6]);
	m_jntPosReachLimit := calcCmdReachLimit();
	m_jntEnableFlag := faultDetect(i_slaveCart.curJntPos);
	FOR i := 5 TO 8 DO 
		m_tarJntPos[i] := LIMIT(GVL_CartMotorParameters.g_minJntPos[i] + m_carJntSoftwareLimit[i], m_trajJntPos[i], GVL_CartMotorParameters.g_maxJntPos[i] - m_carJntSoftwareLimit[i]) ;
		m_jntOTG[i].run(i_targetPos:= m_tarJntPos[i], i_targetVel:= 0.0, o_cmdAcc=> , o_cmdVel=> , o_cmdPos=>m_cmdJntPos[i] );
	END_FOR
END_IF
END_METHOD

METHOD calcCmdReachLimit : vec8b
VAR_INPUT
END_VAR

VAR
	i : INT;
END_VAR

FOR i := 5 TO g_cartJntNum DO
	IF (GVL_CartMotorParameters.g_minJntPos[i] + m_carJntSoftwareLimit[i]) >= m_trajJntPos[i] THEN
		IF (m_tarPosInc[i] - m_lastPosInc[i]) <0 THEN
			m_tarPosInc[i] := m_lastPosInc[i];
		END_IF
		calcCmdReachLimit[i] := TRUE;
	
	ELSIF m_trajJntPos[i]>=(m_maxJntPos[i] - m_carJntSoftwareLimit[i]) THEN
		IF (m_tarPosInc[i] - m_lastPosInc[i]) >0 THEN
			m_tarPosInc[i] := m_lastPosInc[i];
		END_IF
		calcCmdReachLimit[i] := TRUE;
	END_IF
	m_lastPosInc[i] := m_tarPosInc[i];
END_FOR
END_METHOD

METHOD faultDetect : vec8i
VAR_INPUT
	curJntPos : vec8d;
END_VAR
faultDetect[5] := BOOL_TO_INT( NOT SafetyCheck.m_safetyCheckData.m_cartStandColumnErr);
faultDetect[6] := BOOL_TO_INT( NOT SafetyCheck.m_safetyCheckData.m_cartAdjustErr);
faultDetect[7] := BOOL_TO_INT( NOT SafetyCheck.m_safetyCheckData.m_cartAdjustErr);
faultDetect[8] := BOOL_TO_INT( NOT SafetyCheck.m_safetyCheckData.m_cartAdjustErr);

IF SafetyCheck.m_safetyCheckData.m_cartStandColumnErr THEN
	m_trajJntPos[5] :=curJntPos[5];
END_IF
IF SafetyCheck.m_safetyCheckData.m_cartAdjustErr THEN
	m_trajJntPos[6] :=curJntPos[6];
	m_trajJntPos[7] :=curJntPos[7];
	m_trajJntPos[8] :=curJntPos[8];
END_IF
END_METHOD

// override this function in each exact controller
// NOTICE: set joint control mode here, and do some initialization if needed
METHOD PUBLIC init : BOOL
VAR_IN_OUT CONSTANT
	i_slaveCart	:FB_SlaveCart;
END_VAR
VAR_IN_OUT 
	r_cartCtrlCmd :ST_SlaveArmCtrlCmds;
END_VAR
VAR
	i:INT;
END_VAR
// check if to hold the command joint position unchanged
//m_holdLastCmds := checkToHoldLastCmds(i_slaveCart);
m_holdLastCmds := checkToHoldLastCmds(i_slaveCart);
SUPER^.init(i_slaveCart,r_cartCtrlCmd);

m_jntEnableFlag[5] := BOOL_TO_INT( NOT SafetyCheck.m_safetyCheckData.m_cartStandColumnErr);
m_jntEnableFlag[6] := BOOL_TO_INT( NOT SafetyCheck.m_safetyCheckData.m_cartAdjustErr);
m_jntEnableFlag[7] := BOOL_TO_INT( NOT SafetyCheck.m_safetyCheckData.m_cartAdjustErr);
m_jntEnableFlag[8] := BOOL_TO_INT( NOT SafetyCheck.m_safetyCheckData.m_cartAdjustErr);

m_jntOPMode[5]:= DriverOPMode_cspMZ;
m_jntOPMode[6]:= DriverOPMode_Pos;
m_jntOPMode[7]:= DriverOPMode_Pos;
m_jntOPMode[8]:= DriverOPMode_Pos;

m_joystickSignal := g_zeroVec8d;
m_tarPosInc := g_zeroVec8d;
m_trajJntPos := g_zeroVec8d;
m_jntPosReachLimit := g_zeroVec8b;

m_maxJntPos := GVL_CartMotorParameters.g_maxJntPos;
m_maxJntPos[5] := i_slaveCart.m_cartDataFromUI.m_standColumnHightLimit;

m_initActJntPos:=m_cmdJntPos;//i_slaveCart.curJntPos;
m_initActCartPos[6] := (m_initActJntPos[7] + GVL_CartControlParameters.g_curBeamStretchJntInitPos) * SIN(m_initActJntPos[6]);
m_initActCartPos[7] := (m_initActJntPos[7] + GVL_CartControlParameters.g_curBeamStretchJntInitPos) * COS(m_initActJntPos[6]);

FOR i := 1 TO 4 BY 1 DO
	m_jntOTG[i+4].init(i_curCmdPos:= m_cmdJntPos[i+4], i_curCmdVel:= 0, i_maxV:=GVL_CartControlParameters.g_maxJntVel[i+4] , i_maxA:=GVL_CartControlParameters.g_maxJntAcc[i+4] , i_Ts:=g_cartCtrlCycleTime );
END_FOR

m_adjustStartTime := 0;
// update commands to arm
copyCmds(r_cartCtrlCmd);
END_METHOD

PROPERTY jntPosReachLimit : vec8b
GET
jntPosReachLimit := m_jntPosReachLimit;
END_GET
END_PROPERTY

END_FUNCTION_BLOCK

// ---- FBs_CartControlles/FB_CartCtrlRotaOverhang.TcPOU
FUNCTION_BLOCK FB_CartCtrlRotaOverhang EXTENDS FB_CartCtrlBase
VAR_INPUT
END_VAR
VAR_OUTPUT
END_VAR
VAR

	m_actJntPos: Vec8d;
	m_tarJntPos: Vec8d;
	m_cmdJntDir : INT;
	m_rotaAngle:LREAL:=2.5 * g_deg2Rad ;
	m_initJntPos : LREAL;
	m_tarJntInc : LREAL;

	m_carJntSoftwareLimit :ARRAY [5..8] OF LREAL := [0.005, 2*g_deg2Rad, 0.005, 2*g_deg2Rad];
	
	// time threshold to 5-8joint after it's enabled
	m_cartAdjustStartWaitTime :LREAL := 0.2;
	
	//adjust start  time 
	m_adjustStartTime :LREAL;

	m_jntOTG : FB_secOrdTrajFilter;
END_VAR

// override this function in each exact controller
METHOD PROTECTED calcCmdJntPos : BOOL
VAR_IN_OUT CONSTANT
	// slave cart joint data
	i_slaveCart :FB_SlaveCart;
END_VAR

VAR
	i:INT;
END_VAR
//In this method, 8 represents the overhang angle
m_adjustStartTime :=LIMIT(0, m_adjustStartTime + g_cartCtrlCycleTime, 1);
m_actJntPos := i_slaveCart.curJntPos;
IF i_slaveCart.m_rotaOverhangOnFlag = 1 THEN
	m_cmdJntDir := -1;
ELSIF i_slaveCart.m_rotaOverhangOnFlag = 2 THEN
	m_cmdJntDir := 1;
END_IF

IF m_adjustStartTime > m_cartAdjustStartWaitTime THEN
	m_tarJntInc := m_tarJntInc + m_cmdJntDir * m_rotaAngle * g_cartCtrlCycleTime;
	
	m_tarJntPos[8] := LIMIT(GVL_CartMotorParameters.g_minJntPos[8] + m_carJntSoftwareLimit[8], m_initJntPos + m_tarJntInc, GVL_CartMotorParameters.g_maxJntPos[8] - m_carJntSoftwareLimit[8]);

	m_jntOTG.run(i_targetPos:= m_tarJntPos[8], i_targetVel:= 0.0, o_cmdAcc=> , o_cmdVel=> , o_cmdPos=>m_cmdJntPos[8] );
END_IF
END_METHOD

// override this function in each exact controller
// NOTICE: set joint control mode here, and do some initialization if needed
METHOD PUBLIC init : BOOL
VAR_IN_OUT CONSTANT
	i_slaveCart	:FB_SlaveCart;
END_VAR
VAR_IN_OUT 
	r_cartCtrlCmd :ST_SlaveArmCtrlCmds;
END_VAR
VAR
	i:INT;
END_VAR
//m_holdLastCmds := checkToHoldLastCmds(i_slaveCart);
m_holdLastCmds := checkToHoldLastCmds(i_slaveCart);

SUPER^.init(i_slaveCart,r_cartCtrlCmd);

m_jntEnableFlag[8] :=1;

m_jntOPMode[8]:= DriverOPMode_Pos;
m_initJntPos :=m_cmdJntPos[8];
m_tarJntInc := 0;

m_jntOTG.init(i_curCmdPos:= m_cmdJntPos[8], i_curCmdVel:= 0, i_maxV:=GVL_CartControlParameters.g_maxJntVel[8] , i_maxA:=GVL_CartControlParameters.g_maxJntAcc[8] , i_Ts:=g_cartCtrlCycleTime );


m_adjustStartTime := 0;
// update commands to arm
copyCmds(r_cartCtrlCmd);
END_METHOD

END_FUNCTION_BLOCK

// ---- FBs_CartControlles/FB_CartCtrlSlowDown.TcPOU
FUNCTION_BLOCK FB_CartCtrlSlowDown EXTENDS FB_CartCtrlBase
VAR_INPUT
END_VAR
VAR_OUTPUT
END_VAR
VAR

	m_tarPosInc: Vec8d;
	m_trajVel : Vec8d;
	m_initVel : Vec8d;
	m_initPos : Vec8d;
	m_initDec : Vec8d;
	
	//slow down and stop time
	m_incSlowStopTime :LREAL;
	m_slowStopTime :LREAL :=0.5;
	
	// filter cut-off frequency for cart drive force 
	m_cmdJoystickLpfCutoffFreq : LREAL :=8;
	m_cartCtrlFreq :LREAL:=8000;
END_VAR

// override this function in each exact controller
METHOD PROTECTED calcCmdJntPos : BOOL
VAR_IN_OUT CONSTANT
	// slave cart joint data
	i_slaveCart :FB_SlaveCart;
END_VAR

VAR
	i:INT;
END_VAR
//In this method, 5 represents the pillar postion , 6 represents the beam rotation angle ,7 represents the beam stretch position ,8 represents the overhang angle
m_incSlowStopTime :=LIMIT(0, m_incSlowStopTime + g_cartCtrlCycleTime, 1);

FOR i := 1 TO 8 BY 1 DO
	m_trajVel[i] := m_initVel[i] - m_initDec[i] * m_incSlowStopTime;
	IF ABS(m_initVel[i]) < ABS(m_initDec[i]) * m_incSlowStopTime THEN
		m_trajVel[i]:=0;
	END_IF
	m_tarPosInc[i] := m_tarPosInc[i] + m_trajVel[i] * g_cartCtrlCycleTime;
	m_cmdJntPos[i] := m_initPos[i] + m_tarPosInc[i];
END_FOR

IF m_incSlowStopTime >= m_slowStopTime THEN//m_slowStopTime THEN
	m_isFinished := TRUE;
END_IF
END_METHOD

// override this function in each exact controller
// NOTICE: set joint control mode here, and do some initialization if needed
METHOD PUBLIC init : BOOL
VAR_IN_OUT CONSTANT
	i_slaveCart	:FB_SlaveCart;
END_VAR
VAR_IN_OUT 
	r_cartCtrlCmd :ST_SlaveArmCtrlCmds;
END_VAR
m_cmdJntPos:=r_cartCtrlCmd.m_cmdJntPos;
m_initPos := m_cmdJntPos;

m_jntEnableFlag :=r_cartCtrlCmd.m_jntEnableFlag;

m_jntOPMode[5]:= DriverOPMode_cspMZ;
m_jntOPMode[6]:= DriverOPMode_Pos;
m_jntOPMode[7]:= DriverOPMode_Pos;
m_jntOPMode[8]:= DriverOPMode_Pos;

m_trajVel[5] := 0;
m_trajVel[6] := 0;
m_trajVel[7] := 0;
m_trajVel[8] := 0;

m_tarPosInc[5] := 0;
m_tarPosInc[6] := 0;
m_tarPosInc[7] := 0;
m_tarPosInc[8] := 0;


m_incSlowStopTime := 0;

m_initVel[5] := LIMIT(-GVL_CartMotorParameters.g_maxJntVel[5], i_slaveCart.curJntVel[5], GVL_CartMotorParameters.g_maxJntVel[5]);
m_initVel[6] := LIMIT(-GVL_CartMotorParameters.g_maxJntVel[6], i_slaveCart.curJntVel[6], GVL_CartMotorParameters.g_maxJntVel[6]);
m_initVel[7] := LIMIT(-GVL_CartMotorParameters.g_maxJntVel[7], i_slaveCart.curJntVel[7], GVL_CartMotorParameters.g_maxJntVel[7]);
m_initVel[8] := LIMIT(-GVL_CartMotorParameters.g_maxJntVel[8], i_slaveCart.curJntVel[8], GVL_CartMotorParameters.g_maxJntVel[8]);


m_initDec[5] := sign(m_initVel[5])*GVL_CartMotorParameters.g_maxJntVel[5]*2;
m_initDec[6] := sign(m_initVel[6])*GVL_CartMotorParameters.g_maxJntVel[6]*2;
m_initDec[7] := sign(m_initVel[7])*GVL_CartMotorParameters.g_maxJntVel[7]*2;
m_initDec[8] := sign(m_initVel[8])*GVL_CartMotorParameters.g_maxJntVel[8]*2;


m_slowStopTime := 0.5;
// update commands to arm
copyCmds(r_cartCtrlCmd);
END_METHOD

END_FUNCTION_BLOCK

// ---- FBs_CartControlles/FB_CartCtrlStandColuAdjust.TcPOU
FUNCTION_BLOCK FB_CartCtrlStandColuAdjust EXTENDS FB_CartCtrlBase
VAR_INPUT
END_VAR
VAR_OUTPUT
END_VAR
VAR

	m_actJntPos: Vec8d;
	m_tarJntPos : LREAL;
	m_trjJntPos : LREAL;
	m_trjJntInc : LREAL;
	m_lastTrajJntPos : LREAL;
	m_initActJntPos: LREAL;
	m_jntPosReachLimit : Vec8b;
	m_maxJntPos : vec8d;
	m_carJntSoftwareLimit :ARRAY [5..8] OF LREAL := [0.005, 2*g_deg2Rad, 0.005, 2*g_deg2Rad];
	
	// time threshold to 5-8joint after it's enabled
	m_cartAdjustStartWaitTime :LREAL := 0.3;
	
	//adjust start  time 
	m_adjustStartTime :LREAL;
	m_jntOTG : FB_secOrdTrajFilter;
END_VAR

// override this function in each exact controller
METHOD PROTECTED calcCmdJntPos : BOOL
VAR_IN_OUT CONSTANT
	// slave cart joint data
	i_slaveCart :FB_SlaveCart;
END_VAR

VAR
	i:INT;
END_VAR
//In this method, 5 represents the pillar postion , 6 represents the beam rotation angle ,7 represents the beam stretch position ,8 represents the overhang angle
m_adjustStartTime :=LIMIT(0, m_adjustStartTime + g_cartCtrlCycleTime, 1);
m_actJntPos := i_slaveCart.curJntPos;
m_jntEnableFlag[5] := BOOL_TO_INT( NOT SafetyCheck.m_safetyCheckData.m_cartStandColumnErr);

IF m_adjustStartTime > m_cartAdjustStartWaitTime THEN
	m_trjJntInc := m_trjJntInc + (i_slaveCart.m_columnJntVel * g_cartCtrlCycleTime);
	m_trjJntPos := m_initActJntPos + m_trjJntInc;
	m_jntPosReachLimit[5] := calcCmdReachLimit();
	m_tarJntPos := LIMIT(GVL_CartMotorParameters.g_minJntPos[5] + m_carJntSoftwareLimit[5], m_trjJntPos, MAX(m_actJntPos[5],i_slaveCart.m_cartDataFromUI.m_standColumnHightLimit));
	m_jntOTG.run(i_targetPos:= m_tarJntPos, i_targetVel:= 0.0, o_cmdAcc=> , o_cmdVel=> , o_cmdPos=>m_cmdJntPos[5] );
END_IF
END_METHOD

METHOD calcCmdReachLimit : BOOL
VAR_INPUT
END_VAR

VAR
	i : INT;
END_VAR
//IF (GVL_CartMotorParameters.g_minJntPos[5] + m_carJntSoftwareLimit[5]) >= m_trjJntPos OR m_trjJntPos>=(m_maxJntPos[5] - m_carJntSoftwareLimit[5])  THEN
//	calcCmdReachLimit := TRUE;
//END_IF

IF (GVL_CartMotorParameters.g_minJntPos[5] + m_carJntSoftwareLimit[5]) >= m_trjJntPos THEN
	IF (m_trjJntInc - m_lastTrajJntPos) <0 THEN
		m_trjJntInc := m_lastTrajJntPos;
	END_IF
	calcCmdReachLimit := TRUE;

ELSIF m_trjJntPos>=(m_maxJntPos[5] - m_carJntSoftwareLimit[5]) THEN
	IF (m_trjJntInc - m_lastTrajJntPos) >0 THEN
		m_trjJntInc := m_lastTrajJntPos;
	END_IF
	calcCmdReachLimit := TRUE;
END_IF
m_lastTrajJntPos := m_trjJntInc;
END_METHOD

// override this function in each exact controller
// NOTICE: set joint control mode here, and do some initialization if needed
METHOD PUBLIC init : BOOL
VAR_IN_OUT CONSTANT
	i_slaveCart	:FB_SlaveCart;
END_VAR
VAR_IN_OUT 
	r_cartCtrlCmd :ST_SlaveArmCtrlCmds;
END_VAR
VAR
	i:INT;
END_VAR
// check if to hold the command joint position unchanged
//m_holdLastCmds := checkToHoldLastCmds(i_slaveCart);
m_holdLastCmds := checkToHoldLastCmds(i_slaveCart);
SUPER^.init(i_slaveCart,r_cartCtrlCmd);

m_jntEnableFlag[5] := BOOL_TO_INT( NOT SafetyCheck.m_safetyCheckData.m_cartStandColumnErr);
m_jntOPMode[5]:= DriverOPMode_cspMZ;
m_jntPosReachLimit := g_zeroVec8b;
m_maxJntPos[5] := i_slaveCart.m_cartDataFromUI.m_standColumnHightLimit;
m_initActJntPos:=m_cmdJntPos[5];
m_jntOTG.init(i_curCmdPos:= m_cmdJntPos[5], i_curCmdVel:= 0, i_maxV:=GVL_CartControlParameters.g_maxJntVel[5] , i_maxA:=GVL_CartControlParameters.g_maxJntAcc[5] , i_Ts:=g_cartCtrlCycleTime );

m_trjJntInc := 0;
m_adjustStartTime := 0;
// update commands to arm
copyCmds(r_cartCtrlCmd);
END_METHOD

PROPERTY jntPosReachLimit : vec8b
GET
jntPosReachLimit := m_jntPosReachLimit;
END_GET
END_PROPERTY

END_FUNCTION_BLOCK

// ---- AgiMaths/Frames/DHTrans.TcPOU
FUNCTION DHTrans : ST_Frame
VAR_IN_OUT CONSTANT
	// DH parameters: alpha, a, d, theta
	DH :Vec4d;
END_VAR
VAR
END_VAR

DHTrans.m_rot[1,1]:= COS(DH[3]);
DHTrans.m_rot[1,2]:=  -SIN(DH[3]);
DHTrans.m_rot[1,3]:= 0;
DHTrans.m_rot[2,1]:= COS(DH[1])*SIN(DH[3]);
DHTrans.m_rot[2,2]:= COS(DH[1])*COS(DH[3]);
DHTrans.m_rot[2,3]:= -SIN(DH[1]);
DHTrans.m_rot[3,1]:= SIN(DH[1])*SIN(DH[3]);
DHTrans.m_rot[3,2]:= SIN(DH[1])*COS(DH[3]);
DHTrans.m_rot[3,3]:= COS(DH[1]);

DHTrans.m_pos[1]:=DH[2];
DHTrans.m_pos[2]:=-DH[4]*SIN(DH[1]);
DHTrans.m_pos[3]:=DH[4]*COS(DH[1]);

END_FUNCTION

// ---- AgiMaths/Frames/rotX.TcPOU
FUNCTION rotX : mat3d
VAR_INPUT
	i_ang : LREAL;
END_VAR
VAR
	rot :Mat3d := g_eye3d;
END_VAR

rot[2,2]:=COS(i_ang);
rot[3,3]:=rot[2,2];
rot[3,2]:=SIN(i_ang);
rot[2,3]:=-rot[3,2];
rotX:=rot;

END_FUNCTION

// ---- AgiMaths/MatrixLib/invMat7.TcPOU
FUNCTION invMat7 : bool
VAR_IN_OUT CONSTANT
	mat :Mat7d;
END_VAR
VAR_IN_OUT
	invMat : Mat7d;
END_VAR
VAR
	n:INT:=7;
	m:INT:=1;
	b :ARRAY[1..7] OF LREAL := [7(0)];
	indxc,indxr, ipiv:ARRAY[1..7] OF INT := [7(0)];

	
	i,icol, irow, j,k,l,ll: INT;
	big, dum, pivinv,tmp: LREAL;
END_VAR

invMat := mat;
FOR i:=1 TO n DO   
    big:=0.0;
    FOR j:=1 TO n DO  
        IF (ipiv[j] <> 1) THEN
            FOR k:=1 TO n DO 
                IF (ipiv[k] = 0) THEN
                    IF (ABS(invMat[j,k]) >= big) THEN
                        big:=ABS(invMat[j,k]);
                        irow:=j;
                        icol:=k;
                    END_IF
                END_IF
            END_FOR
        END_IF
    END_FOR
    ipiv[icol]:=ipiv[icol]+1;
    
    IF (irow <> icol) THEN
        FOR l:=1 TO n DO 
            tmp:=invMat[irow,l];
            invMat[irow,l]:=invMat[icol,l];
            invMat[icol,l]:=tmp;
        END_FOR
 (*       FOR  l:=1 TO m DO  
            tmp:=b[irow,l];
            b[irow,l]:=b[icol,l];
            b[icol,l]:=tmp;
        END_FOR*)
    END_IF
	
    indxr[i]:=irow; 
    indxc[i]:=icol;
	
     IF ABS(invMat[icol,icol]) < g_smallNum THEN 
          invMat7:=FALSE;
		  RETURN;
    END_IF
	
    pivinv:=1.0/invMat[icol,icol];
    invMat[icol,icol]:=1.0;
    FOR l:=1 TO n DO  
        invMat[icol,l] := invMat[icol,l]*pivinv;
    END_FOR
 (*   FOR l:=1 TO m DO 
        b[icol,l] := b[icol,l]*pivinv;
    END_FOR*)
    FOR ll:=1 TO n DO  
        IF (ll <> icol) THEN 
            dum:=invMat[ll,icol];
            invMat[ll,icol]:=0.0;
            FOR l:=1 TO n DO  
                invMat[ll,l]:=invMat[ll,l] - invMat[icol,l]*dum;
            END_FOR
   (*         FOR l:=1 TO m DO  
                b[ll,l]:=b[ll,l] - b[icol,l]*dum;
            END_FOR*)
        END_IF
    END_FOR

END_FOR


FOR l:=n-1 TO 1 BY -1 DO 
    IF (indxr[l] <> indxc[l]) THEN
        FOR k:=1 TO n DO
            tmp:=invMat[k,indxr[l]];
            invMat[k,indxr[l]]:=invMat[k,indxc[l]];
            invMat[k,indxc[l]]:=tmp;
        END_FOR
    END_IF
END_FOR

invMat7:=TRUE;

END_FUNCTION

// ---- AgiMaths/MatrixLib/matAdd.TcPOU
// C = A + B;
FUNCTION matAdd : BOOL
VAR_IN_OUT CONSTANT
	matA :ARRAY[*,*] OF LREAL;
	matB :ARRAY[*,*] OF LREAL;
END_VAR

VAR_IN_OUT 
	matC :ARRAY[*,*] OF LREAL;
END_VAR

VAR
	m,n :DINT;
	i,j, k :DINT;
 
END_VAR

m:=UPPER_BOUND(matC,1);
n:= UPPER_BOUND(matC,2);
FOR i:=1 TO m DO
	FOR j:=1 TO n DO
		matC[i,j]:=matA[i,j] + matB[i,j];
	END_FOR
END_FOR

END_FUNCTION

// ---- FBs_Auxiliary/FB_IOCheck.TcPOU
// return true if IO is triggerd for a set time period
FUNCTION_BLOCK FB_IOCheck
VAR
	// IO type, 0- normally-opend IO; 1- normally-closed IO
	m_IOType :INT :=0;
	
	// counts after IO  is triggerd
	m_IOOnCounts :INT;
	
	// counts threshold indicating IO is trully triggerd
	m_IOOnCountThres :INT :=100;
END_VAR

METHOD check : BOOL
VAR_INPUT
	IOValue :BOOL;
END_VAR
IF (0=m_IOType and IOValue) OR (1=m_IOType AND NOT(IOValue)) THEN
	m_IOOnCounts := MIN(m_IOOnCounts +1, m_IOOnCountThres);
ELSE
	 m_IOOnCounts :=0;
END_IF

check:=m_IOOnCounts>=m_IOOnCountThres;
END_METHOD

METHOD init : BOOL
VAR_INPUT
	i_IOType :INT;
	i_triggerCounts:INT;
END_VAR
m_IOType:=i_IOType;
m_IOOnCountThres := i_triggerCounts;
END_METHOD

END_FUNCTION_BLOCK

// ---- FBs_Auxiliary/FB_setupAdjustDetect.TcPOU
FUNCTION_BLOCK FB_setupAdjustDetect
VAR_INPUT
END_VAR
VAR_OUTPUT
END_VAR
VAR
	m_manualAdjustOnCounts :INT :=0;
	m_adjustOnCountThres :INT :=50;
END_VAR

// check if instrument is on
METHOD run : BOOL
VAR_INPUT
	IOValue :UDINT;
END_VAR

VAR_OUTPUT
	
END_VAR
// manuel adjust io is 4th bit 
IF 16=(IOValue AND 10#16) THEN
	m_manualAdjustOnCounts :=MIN(m_manualAdjustOnCounts +1,m_adjustOnCountThres);
ELSE
	m_manualAdjustOnCounts :=0;
END_IF

run := m_manualAdjustOnCounts >= m_adjustOnCountThres;
END_METHOD

END_FUNCTION_BLOCK

// ---- FBs_Auxiliary/FB_setupJnt5AdjustDetect.TcPOU
FUNCTION_BLOCK FB_setupJnt5AdjustDetect
VAR_INPUT
END_VAR
VAR_OUTPUT
END_VAR
VAR
	m_pAutoAdjustOnCounts :INT :=0;
	m_nAutoAdjustOnCounts :INT :=0;
	m_adjustOnCountThres :INT :=50;
END_VAR

METHOD run : INT
VAR_INPUT
	IOValue :UDINT;
END_VAR

VAR_OUTPUT
	
END_VAR
// joint3 positive auto adjust is 3th bit
IF 4=(IOValue AND 10#4) THEN
	m_pAutoAdjustOnCounts :=MIN(m_pAutoAdjustOnCounts +1,m_adjustOnCountThres);
ELSE
	m_pAutoAdjustOnCounts :=0;
END_IF

// joint3 negative auto adjust is 2th bit
IF 2=(IOValue AND 10#2) THEN
	m_nAutoAdjustOnCounts :=MIN(m_nAutoAdjustOnCounts +1,m_adjustOnCountThres);
ELSE
	m_nAutoAdjustOnCounts :=0;
END_IF

IF m_pAutoAdjustOnCounts >= m_adjustOnCountThres THEN
	run :=1;
ELSIF m_nAutoAdjustOnCounts >= m_adjustOnCountThres THEN
	run := -1;
ELSE 
	run :=0;
END_IF
END_METHOD

END_FUNCTION_BLOCK

// ---- FBs_BasicControllers/FB_dither.TcPOU
FUNCTION_BLOCK FB_dither
VAR_INPUT
END_VAR
VAR_OUTPUT
END_VAR
VAR
	// dithering signal type
	// 1: square
	m_type:INT := 1;
	
	// dithering amplitude
	m_amplitude:LREAL;
	
	// dithering frequency
	m_frequency :LREAL;
	
	// time step
	m_timeStep :LREAL;
	
	// time period
	m_timePeriod:LREAL:=0.0;
END_VAR

METHOD init : BOOL
VAR_INPUT
	i_type:INT;
	i_timeStep:LREAL;
	i_amp:LREAL;
	i_freq:LREAL;
END_VAR
m_type:=i_type;
m_timeStep:=i_timeStep;
m_amplitude:=i_amp;
m_frequency:= i_freq;
m_timePeriod:=0;
END_METHOD

METHOD run : LREAL
VAR_INPUT
END_VAR
VAR
	tmpVar :LREAL;
END_VAR
m_timePeriod := m_timePeriod+ m_timeStep;
run:=0;

CASE m_type OF
	// sin
	1:
		run := m_amplitude*SIN(2*pi*m_frequency * m_timePeriod);
	// square
	2:
		tmpVar := SIN(2*pi*m_frequency * m_timePeriod);
		run:= sign(tmpVar) * m_amplitude;
	
END_CASE
END_METHOD

END_FUNCTION_BLOCK

// ---- FBs_BasicControllers/FBMacroJntControl.TcPOU
// Author: Feijian Ni
// Date: 2023.11.22
FUNCTION_BLOCK FBMacroJntControl
VAR_INPUT
END_VAR
VAR_OUTPUT
END_VAR
VAR
	//TODO: move to GVLs 
	// control paramters
	m_macroJntKp:ARRAY[1..3] OF LREAL:=[1200,10,10];
	m_macroJntKd:ARRAY[1..4] OF LREAL:=[100,1.0,1.0];
	m_macroJntKi:ARRAY[1..4] OF LREAL:=[3000,0,0,0];
	m_macroJntKiLimit:ARRAY[1..4] OF LREAL:=[3(1500.0)];
	m_macroJnttrlLimit:ARRAY[1..4] OF LREAL:=[3(3500.0)];
	m_jntTargetPosLpfCutoffFreq:LREAL:=10;
	m_curJntVelLpfCutoffFreq:LREAL:=30;
	
	// filter for target joint position
	m_cmdPosLpf:ARRAY[1..3] OF FBLowPassFilter;
	
	// filter for current joint velocity
	m_curJntVelLpf:ARRAY[1..3] OF FBLowPassFilter;
	
	// max command joint velocity
	m_maxJntVel:ARRAY[1..3] OF LREAL:=[1.5, 0.1, 0.1];
	
	// arm index for grip control
	m_armIdx:INT;
	
	// final target macro joint position
	m_targetJntPos:ARRAY[1..3] OF LREAL;
	
	// position tracking error
	m_posErr:ARRAY[1..3] OF LREAL;
	
	// max position error for safety check
	m_safetyPosErr:ARRAY[1..3] OF LREAL:=[5.0*pi/180,5.0*pi/180,0.01];
	
	// command macro joint position and veloicty for next cycle
	m_cmdJntPos:ARRAY[1..3] OF LREAL;
	m_cmdJntVel:ARRAY[1..3] OF LREAL;

	// current  macro joint position and veloicty for next cycle
	m_curJntPos:ARRAY[1..3] OF LREAL;
	m_curJntVel:ARRAY[1..3] OF LREAL;
	
	// PID for joint position
	m_jntPIDCtrl:ARRAY[1..3] OF FBPID;
	m_cmdJntTrq:ARRAY[1..3] OF LREAL;
	
END_VAR

METHOD init : BOOL
VAR_INPUT
	i_armIdx:INT;
END_VAR

VAR
	i,j:INT;
	currentRatioMotor2Jnt:LREAL;
END_VAR
m_armIdx:=i_armIdx;

// get current instrument orientation
m_curJntPos[1]:=Robot_Status.Robot_Current_DH_Joint_Position_M3[m_armIdx].q1;
m_curJntPos[2]:=Robot_Status.Robot_Current_DH_Joint_Position_M3[m_armIdx].q2;
m_curJntPos[3]:=Robot_Status.Robot_Current_DH_Joint_Position_M3[m_armIdx].q3;
FOR i:=1 TO 3  DO 
	m_targetJntPos[i]:=m_curJntPos[i];
	m_cmdJntPos[i]:=m_curJntPos[i];
	m_cmdJntVel[i]:=0;
	m_curJntVel[i]:=0;
END_FOR

